	garr_betriebsmeldungen[st_config.i16_meld_startindex + 0] := fb_ton_abfrage_wt_auf_beladepos.Q;
	garr_betriebsmeldungen[st_config.i16_meld_startindex + 1] := fb_ton_warte_auf_wt_an_stopper.Q;
	garr_betriebsmeldungen[st_config.i16_meld_startindex + 2] := FALSE;
	garr_betriebsmeldungen[st_config.i16_meld_startindex + 3] := FALSE;
	garr_betriebsmeldungen[st_config.i16_meld_startindex + 4] := FALSE;
	garr_betriebsmeldungen[st_config.i16_meld_startindex + 5] := FALSE;
	garr_betriebsmeldungen[st_config.i16_meld_startindex + 6] := FALSE;
	garr_betriebsmeldungen[st_config.i16_meld_startindex + 7] := FALSE;
	garr_betriebsmeldungen[st_config.i16_meld_startindex + 8] := FALSE;
	garr_betriebsmeldungen[st_config.i16_meld_startindex + 9] := FALSE;
	garr_betriebsmeldungen[st_config.i16_meld_startindex + 10] := FALSE;
	garr_betriebsmeldungen[st_config.i16_meld_startindex + 11] := FALSE;
	garr_betriebsmeldungen[st_config.i16_meld_startindex + 12] := FALSE;
	garr_betriebsmeldungen[st_config.i16_meld_startindex + 13] := FALSE;
	garr_betriebsmeldungen[st_config.i16_meld_startindex + 14] := FALSE;
	garr_betriebsmeldungen[st_config.i16_meld_startindex + 15] := FALSE;
	garr_betriebsmeldungen[st_config.i16_meld_startindex + 16] := FALSE;
	garr_betriebsmeldungen[st_config.i16_meld_startindex + 17] := FALSE;
	garr_betriebsmeldungen[st_config.i16_meld_startindex + 18] := FALSE;
	garr_betriebsmeldungen[st_config.i16_meld_startindex + 19] := FALSE;
END_IF
END_PROGRAM

(* POU Gemeinsamkeiten17xx/WT Transport/ST_Hublift_links, ST *)
PROGRAM ST_Hublift_links
VAR_INPUT
	st_config							: struct_config;
	st_ctrl_in							: struct_ctrl_in;
	e_station_nachher_in_erlaubnis		: BOOL := FALSE;
	e_station_nachher_in_angekommen	: BOOL := FALSE;
END_VAR
VAR_IN_OUT
	st_visu							: struct_visu;
END_VAR
VAR_OUTPUT
	st_ctrl_out						: struct_ctrl_out;
	a_station_nachher_out_anforderung	: BOOL := FALSE;
	a_station_nachher_out_abgegeben	: BOOL := FALSE;
END_VAR
VAR
	fb_ton_wz						: TON;
	fb_ton_uez						: TON;
	tb_ton_wt_anwesend				: TON;
	fb_ton_quitt						: TON;
	fb_r_trig_start						: R_TRIG;
	fb_state_entry						: ST_StateEntry;
	sm_kein_wt_anwesend				: BOOL := FALSE;
	sm_keine_busverbindung			: BOOL := FALSE;
	sm_schiebetuere_nicht_geschlossen	: BOOL := FALSE;

	e_sensor_wt_anwesend			AT %I* : BOOL;
	e_sensor_wt_von_fb_eingezogen	AT %I* : BOOL;
	e_wc_state						AT%I*: BOOL;	(* 0=Data valid, 1=Data invalid *)

	e_schiebetuere_geschlossen			AT %I* : BOOL;
	a_lampe_erlaubnis_schiebetuere_oeffnen		AT %Q* : BOOL;	(* Wenn Lampe TRUE dann darf der Bediener die Schiebetüre öffnen *)
END_VAR
(* Zeiten *)
fb_ton_wz(IN:= , PT:= , Q=>  , ET=> );
fb_ton_uez(IN:= , PT:= , Q=>  , ET=> );
tb_ton_wt_anwesend(IN:=e_sensor_wt_anwesend , PT:= t#500ms, Q=>  , ET=> );
fb_ton_quitt(IN:= , PT:= t#100ms, Q=> , ET=> );

(* Flanken *)
fb_r_trig_start(CLK:=ST_Euchner_Handbedienpult.b_Taste_Power , Q=>);

(* Toplevel *)
IF fb_state_entry.i16_next_step > INIT AND fb_state_entry.i16_next_step < FEHLER THEN
	IF fb_state_entry.i16_next_step < STOP THEN
		IF st_ctrl_in.b_stop THEN
			fb_state_entry.i16_next_step := STOP;
		END_IF
	END_IF

	(* Allgemeine Fehler *)
	IF 	st_config.b_station_aktiv AND NOT st_config.b_station_in_simulation AND
		(zyl_hublift_links_lift.st_ctrl.out.b_fehler OR
		zyl_hublift_links_wt_einzug.st_ctrl.out.b_fehler OR
		zyl_hublift_links_wt_klinke.st_ctrl.out.b_fehler OR
		zyl_hublift_links_stopper.st_ctrl.out.b_fehler OR
		zyl_hublift_links_eingriffschutz.st_ctrl.out.b_fehler) THEN
			fb_state_entry.i16_next_step := FEHLER;

	(* Zylinder im Handbetrieb *)
	ELSIF gi16_betriebsart = HAND AND st_config.b_station_aktiv AND NOT st_config.b_station_in_simulation AND
		((st_visu.st_zyl.i16_nr_zyl_im_handbetrieb = zyl_hublift_links_lift.fb.st_config.i16_identnummer) OR
		(st_visu.st_zyl.i16_nr_zyl_im_handbetrieb = zyl_hublift_links_wt_einzug.fb.st_config.i16_identnummer) OR
		(st_visu.st_zyl.i16_nr_zyl_im_handbetrieb = zyl_hublift_links_wt_klinke.fb.st_config.i16_identnummer) OR
		(st_visu.st_zyl.i16_nr_zyl_im_handbetrieb = zyl_hublift_links_stopper.fb.st_config.i16_identnummer)  OR
		(st_visu.st_zyl.i16_nr_zyl_im_handbetrieb = zyl_hublift_links_eingriffschutz.fb.st_config.i16_identnummer) ) THEN
			fb_state_entry.i16_next_step := FEHLER;
	END_IF
END_IF

(* ==================================Schrittkette================================ *)
fb_state_entry(
	i16_next_step:= ,
	i16_pos:= 1,
	s_debugtext:= ,
	E=> ,
	X=> ,
	i16_step=> ,
	i16_last_step=> );

CASE fb_state_entry.i16_step OF
(*=======================================================*)
	INIT_OBJ:
		IF st_config.b_config_fertig THEN
			fb_state_entry.i16_next_step := INIT;
		END_IF

(*=======================================================*)
	INIT:
		IF fb_state_entry.E THEN
			fb_ton_wz.IN := FALSE;
			fb_ton_uez.IN	:= FALSE;
			fb_ton_quitt.IN := FALSE;
			sm_kein_wt_anwesend	:= FALSE;
			sm_keine_busverbindung := FALSE;
			sm_schiebetuere_nicht_geschlossen := FALSE;
			a_station_nachher_out_anforderung := FALSE;
			a_station_nachher_out_abgegeben := FALSE;
			a_lampe_erlaubnis_schiebetuere_oeffnen := FALSE;
			st_ctrl_out.b_fehler := FALSE;
			st_ctrl_out.b_bereit := FALSE;
			st_ctrl_out.b_fertig := FALSE;
			st_ctrl_out.b_kontroller_start := FALSE;
			zyl_hublift_links_lift.st_ctrl.in.b_einfahren := FALSE;
			zyl_hublift_links_lift.st_ctrl.in.b_ausfahren := FALSE;
			zyl_hublift_links_wt_einzug.st_ctrl.in.b_einfahren := FALSE;
			zyl_hublift_links_wt_einzug.st_ctrl.in.b_ausfahren := FALSE;
			zyl_hublift_links_wt_klinke.st_ctrl.in.b_einfahren := FALSE;
			zyl_hublift_links_wt_klinke.st_ctrl.in.b_ausfahren := FALSE;
			zyl_hublift_links_stopper.st_ctrl.in.b_einfahren := FALSE;
			zyl_hublift_links_stopper.st_ctrl.in.b_ausfahren := FALSE;
			zyl_hublift_links_eingriffschutz.st_ctrl.in.b_einfahren := FALSE;
			zyl_hublift_links_eingriffschutz.st_ctrl.in.b_ausfahren := FALSE;
		END_IF

		(*-----------------------Weiterschaltbedingungen----------------------------*)
		IF st_ctrl_in.b_init THEN
			zyl_hublift_links_lift.st_ctrl.in.b_quittieren := FALSE;
			zyl_hublift_links_wt_einzug.st_ctrl.in.b_quittieren := FALSE;
			zyl_hublift_links_wt_klinke.st_ctrl.in.b_quittieren := FALSE;
			zyl_hublift_links_stopper.st_ctrl.in.b_quittieren := FALSE;
			zyl_hublift_links_eingriffschutz.st_ctrl.in.b_quittieren := FALSE;

			IF st_config.b_station_aktiv AND NOT st_config.b_station_in_simulation AND gst_datensatz.st_md.b_wt_transport_aktiv THEN
				fb_state_entry.i16_next_step := 15;
			ELSE
				fb_state_entry.i16_next_step := BEREIT;
			END_IF
		END_IF

(*=======================================================*)
	15: (* Prüfe, ob Busverbindung vorhanden ist *)

		(*-----------------------Weiterschaltbedingungen----------------------------*)
		IF e_wc_state THEN
			sm_keine_busverbindung := TRUE;
			fb_state_entry.i16_next_step := FEHLER;
		ELSE
			fb_state_entry.i16_next_step := 18;
		END_IF

(*=======================================================*)
	18: (* Prüfe, ob Eingriffschutz geschlossen ist *)

		(*-----------------------Weiterschaltbedingungen----------------------------*)
		IF NOT e_schiebetuere_geschlossen THEN
			sm_schiebetuere_nicht_geschlossen := TRUE;
			fb_state_entry.i16_next_step := FEHLER;
		ELSE
			fb_state_entry.i16_next_step := 20;
		END_IF

(*=======================================================*)
	20: (* Initialisierung: Stopper ausfahren *)
		IF fb_state_entry.E THEN
			zyl_hublift_links_stopper.st_ctrl.in.b_ausfahren := TRUE;
		END_IF

		(*-----------------------Weiterschaltbedingungen----------------------------*)
		IF zyl_hublift_links_stopper.st_ctrl.out.b_ausgefahren THEN
			zyl_hublift_links_stopper.st_ctrl.in.b_ausfahren := FALSE;
			fb_state_entry.i16_next_step := 30;
		END_IF

(*=======================================================*)
	30: (* Initialisierung: Abfrage auf WT *)
		IF tb_ton_wt_anwesend.Q THEN
		(* WT anwesend *)
			IF zyl_hublift_links_lift.fb.e_sensor1_eingefahren THEN
			(* Hublift unten *)
				fb_state_entry.i16_next_step := 120;
			ELSE
			(* Hublift oben *)
				fb_state_entry.i16_next_step := 155;
			END_IF
		ELSE
		(* Kein WT vorhanden oder vielleicht steht einer am Stopper *)
			fb_state_entry.i16_next_step := 40;
		END_IF

(*=======================================================*)
	40: (* Initialisierung: Klinke einfahren *)
		IF fb_state_entry.E THEN
			zyl_hublift_links_wt_klinke.st_ctrl.in.b_einfahren := TRUE;
		END_IF

		(*-----------------------Weiterschaltbedingungen----------------------------*)
		IF zyl_hublift_links_wt_klinke.st_ctrl.out.b_eingefahren THEN
			zyl_hublift_links_wt_klinke.st_ctrl.in.b_einfahren := FALSE;
			IF zyl_hublift_links_lift.fb.e_sensor1_eingefahren THEN
			(* Hublift unten *)
				fb_state_entry.i16_next_step := 70;
			ELSE
			(* Hublift oben *)
				fb_state_entry.i16_next_step := 50;
			END_IF
		END_IF

(*=======================================================*)
	50: (* Initialisierung: WT-Einzug einfahren *)
		IF fb_state_entry.E THEN
			zyl_hublift_links_wt_einzug.st_ctrl.in.b_einfahren := TRUE;
		END_IF

		(*-----------------------Weiterschaltbedingungen----------------------------*)
		IF zyl_hublift_links_wt_einzug.st_ctrl.out.b_eingefahren THEN
			zyl_hublift_links_wt_einzug.st_ctrl.in.b_einfahren := FALSE;
			fb_state_entry.i16_next_step := 60;
		END_IF

(*=======================================================*)
	60: (* Initialisierung: Lift einfahren *)
		IF fb_state_entry.E THEN
			zyl_hublift_links_lift.st_ctrl.in.b_einfahren := TRUE;
		END_IF

		(*-----------------------Weiterschaltbedingungen----------------------------*)
		IF zyl_hublift_links_lift.st_ctrl.out.b_eingefahren THEN
			zyl_hublift_links_lift.st_ctrl.in.b_einfahren := FALSE;
			fb_state_entry.i16_next_step := 70;
		END_IF

(*=======================================================*)
	70: (* WT-Einzug ausfahren *)
		IF fb_state_entry.E THEN
			zyl_hublift_links_wt_einzug.st_ctrl.in.b_ausfahren := TRUE;
		END_IF

		(*-----------------------Weiterschaltbedingungen----------------------------*)
		IF zyl_hublift_links_wt_einzug.st_ctrl.out.b_ausgefahren THEN
			zyl_hublift_links_wt_einzug.st_ctrl.in.b_ausfahren := FALSE;
			fb_state_entry.i16_next_step := 80;
		END_IF

(*=======================================================*)
	80: (* Initialisierung: Stopper einfahren *)
		IF fb_state_entry.E THEN
			zyl_hublift_links_stopper.st_ctrl.in.b_einfahren := TRUE;
		END_IF

		(*-----------------------Weiterschaltbedingungen----------------------------*)
		IF zyl_hublift_links_stopper.st_ctrl.out.b_eingefahren THEN
			zyl_hublift_links_stopper.st_ctrl.in.b_einfahren := FALSE;
			fb_state_entry.i16_next_step := 90;
		END_IF

(*=======================================================*)
	90: (* Eingriffschutz ausfahren*)
		IF fb_state_entry.E THEN
			zyl_hublift_links_eingriffschutz.st_ctrl.in.b_ausfahren := TRUE;
		END_IF

		(*-----------------------Weiterschaltbedingungen----------------------------*)
		IF zyl_hublift_links_eingriffschutz.st_ctrl.out.b_ausgefahren THEN
			zyl_hublift_links_eingriffschutz.st_ctrl.in.b_ausfahren := FALSE;
			fb_state_entry.i16_next_step := BEREIT;
		END_IF

(*=======================================================*)
	BEREIT:
		IF fb_state_entry.E THEN
			st_ctrl_out.b_bereit := TRUE;
		END_IF

		(*-----------------------Weiterschaltbedingungen----------------------------*)
		IF st_config.b_station_aktiv AND NOT st_config.b_station_in_simulation AND gst_datensatz.st_md.b_wt_transport_aktiv THEN
			(* Hublift und WT Transport aktiv *)
			fb_state_entry.i16_next_step := 110;
		ELSIF NOT st_config.b_station_aktiv AND st_config.b_station_in_simulation AND gst_datensatz.st_md.b_wt_transport_aktiv THEN
			(* Simulation des Hubliftes *)
			fb_state_entry.i16_next_step := 160;
		ELSE
			;(* Hublift und WT Transport NICHT aktiv *)
		END_IF

(*=======================================================*)
	110:	(* Warte bis der WT angekommen ist *)

		(*-----------------------Weiterschaltbedingungen----------------------------*)
		IF tb_ton_wt_anwesend.Q THEN
			fb_state_entry.i16_next_step := 120;
		END_IF

(*=======================================================*)
	120: (* Klinke ausfahren -> WT einhaken*)
		IF fb_state_entry.E THEN
			zyl_hublift_links_wt_klinke.st_ctrl.in.b_ausfahren := TRUE;
		END_IF

		(*-----------------------Weiterschaltbedingungen----------------------------*)
		IF zyl_hublift_links_wt_klinke.st_ctrl.out.b_ausgefahren AND
			e_sensor_wt_anwesend THEN
			zyl_hublift_links_wt_klinke.st_ctrl.in.b_ausfahren := FALSE;
			fb_state_entry.i16_next_step := 130;
		END_IF

(*=======================================================*)
	130: (* WT-Einzug einfahren und Stopper bei Signal ausfahren *)
		IF fb_state_entry.E THEN
			zyl_hublift_links_wt_einzug.st_ctrl.in.b_einfahren := TRUE;
		END_IF

		(*-----------------------Weiterschaltbedingungen----------------------------*)
		IF 	e_sensor_wt_von_fb_eingezogen OR
			zyl_hublift_links_wt_einzug.st_ctrl.out.b_eingefahren THEN
				zyl_hublift_links_stopper.st_ctrl.in.b_ausfahren := TRUE;
				fb_state_entry.i16_next_step := 140;
		END_IF

(*=======================================================*)
	140: (* WT-Einzug ist eingefahren und Stopper ist ausgefahren *)

		(*-----------------------Weiterschaltbedingungen----------------------------*)
		IF 	zyl_hublift_links_stopper.st_ctrl.out.b_ausgefahren AND
			zyl_hublift_links_wt_einzug.st_ctrl.out.b_eingefahren AND
			e_sensor_wt_anwesend THEN
				zyl_hublift_links_stopper.st_ctrl.in.b_ausfahren := FALSE;
				zyl_hublift_links_wt_einzug.st_ctrl.in.b_einfahren := FALSE;
				fb_state_entry.i16_next_step := 150;
		END_IF

(*=======================================================*)
	150: (* WT mit Lift anheben *)
		IF fb_state_entry.E THEN
			zyl_hublift_links_lift.st_ctrl.in.b_ausfahren := TRUE;
		END_IF

		(*-----------------------Weiterschaltbedingungen----------------------------*)
		IF zyl_hublift_links_lift.st_ctrl.out.b_ausgefahren THEN
			zyl_hublift_links_lift.st_ctrl.in.b_ausfahren := FALSE;
			fb_state_entry.i16_next_step := 155;
		END_IF

(*=======================================================*)
	155: (* Warte auf Simulation oder Taste_Power *)
		IF fb_state_entry.E THEN
			a_lampe_erlaubnis_schiebetuere_oeffnen := TRUE;
		END_IF

		(*-----------------------Weiterschaltbedingungen----------------------------*)
		IF st_config.b_station_in_simulation OR
			(fb_r_trig_start.Q AND e_schiebetuere_geschlossen) THEN
			fb_state_entry.i16_next_step := 160;
		END_IF

		IF fb_state_entry.X THEN
			a_lampe_erlaubnis_schiebetuere_oeffnen := FALSE;
		END_IF

(*=======================================================*)
	160: (* Warte auf Folgestation *)
		IF fb_state_entry.E THEN
			st_ctrl_out.b_bereit := TRUE;
			a_station_nachher_out_anforderung := TRUE;
		END_IF

		(*-----------------------Weiterschaltbedingungen----------------------------*)
		IF  e_station_nachher_in_erlaubnis AND NOT fb_state_entry.E THEN
			a_station_nachher_out_anforderung := FALSE;
			IF st_config.b_station_in_simulation THEN
				fb_state_entry.i16_next_step := 180;
			ELSE
				IF e_sensor_wt_anwesend THEN
					fb_state_entry.i16_next_step := 165;
				ELSE
					fb_state_entry.i16_next_step := 190;
				END_IF
			END_IF
		END_IF

(*=======================================================*)
	165: (* Eingriffschutz einfahren*)
		IF fb_state_entry.E THEN
			zyl_hublift_links_eingriffschutz.st_ctrl.in.b_einfahren := TRUE;
		END_IF

		(*-----------------------Weiterschaltbedingungen----------------------------*)
		IF zyl_hublift_links_eingriffschutz.st_ctrl.out.b_eingefahren THEN
			zyl_hublift_links_eingriffschutz.st_ctrl.in.b_einfahren := FALSE;
			fb_state_entry.i16_next_step := 170;
		END_IF

(*=======================================================*)
	170: (* WT-Einzug ausfahren und Klinke einfahren und WT aushaken *)
		IF fb_state_entry.E THEN
			zyl_hublift_links_wt_einzug.st_ctrl.in.b_ausfahren := TRUE;
			zyl_hublift_links_wt_klinke.st_ctrl.in.b_einfahren := TRUE;
			st_ctrl_out.b_kontroller_start := TRUE;
		END_IF

		(*-----------------------Weiterschaltbedingungen----------------------------*)
		IF 	zyl_hublift_links_wt_einzug.st_ctrl.out.b_ausgefahren AND
			zyl_hublift_links_wt_klinke.st_ctrl.out.b_eingefahren
			THEN
				st_ctrl_out.b_kontroller_start := FALSE;
				zyl_hublift_links_wt_einzug.st_ctrl.in.b_ausfahren := FALSE;
				zyl_hublift_links_wt_klinke.st_ctrl.in.b_einfahren := FALSE;
				fb_state_entry.i16_next_step := 180;
		END_IF

(*=======================================================*)
	180:	(* Warte bis WT angekommen ist *)
		IF fb_state_entry.E THEN
			a_station_nachher_out_abgegeben := TRUE;
		END_IF

		(*-----------------------Weiterschaltbedingungen----------------------------*)
		IF e_station_nachher_in_angekommen THEN
			a_station_nachher_out_abgegeben := FALSE;
			IF st_config.b_station_in_simulation THEN
				fb_state_entry.i16_next_step := BEREIT;
			ELSE
				fb_state_entry.i16_next_step := 185;
			END_IF
		END_IF

(*=======================================================*)
	185: (* Eingriffschutz ausfahren*)
		IF fb_state_entry.E THEN
			zyl_hublift_links_eingriffschutz.st_ctrl.in.b_ausfahren := TRUE;
		END_IF

		(*-----------------------Weiterschaltbedingungen----------------------------*)
		IF zyl_hublift_links_eingriffschutz.st_ctrl.out.b_ausgefahren THEN
			zyl_hublift_links_eingriffschutz.st_ctrl.in.b_ausfahren := FALSE;
			fb_state_entry.i16_next_step := 190;
		END_IF

(*=======================================================*)
	190: (* Klinke einfahren*)
		IF fb_state_entry.E THEN
			zyl_hublift_links_wt_klinke.st_ctrl.in.b_einfahren := TRUE;
		END_IF

		(*-----------------------Weiterschaltbedingungen----------------------------*)
		IF zyl_hublift_links_wt_klinke.st_ctrl.out.b_eingefahren THEN
			zyl_hublift_links_wt_klinke.st_ctrl.in.b_einfahren := FALSE;
			fb_state_entry.i16_next_step := 200;
		END_IF

(*=======================================================*)
	200: (* WT-Einzug einfahren  *)
		IF fb_state_entry.E THEN
			zyl_hublift_links_wt_einzug.st_ctrl.in.b_einfahren := TRUE;
		END_IF

		(*-----------------------Weiterschaltbedingungen----------------------------*)
		IF zyl_hublift_links_wt_einzug.st_ctrl.out.b_eingefahren THEN
			zyl_hublift_links_wt_einzug.st_ctrl.in.b_einfahren := FALSE;
			fb_state_entry.i16_next_step := 210;
		END_IF

(*=======================================================*)
	210: (*  Lift einfahren *)
		IF fb_state_entry.E THEN
			zyl_hublift_links_lift.st_ctrl.in.b_einfahren := TRUE;
		END_IF

		(*-----------------------Weiterschaltbedingungen----------------------------*)
		IF zyl_hublift_links_lift.st_ctrl.out.b_eingefahren THEN
			zyl_hublift_links_lift.st_ctrl.in.b_einfahren := FALSE;
			fb_state_entry.i16_next_step := 220;
		END_IF

(*=======================================================*)
	220: (* WT-Einzug ausfahren  *)
		IF fb_state_entry.E THEN
			zyl_hublift_links_wt_einzug.st_ctrl.in.b_ausfahren := TRUE;
		END_IF

		(*-----------------------Weiterschaltbedingungen----------------------------*)
		IF zyl_hublift_links_wt_einzug.st_ctrl.out.b_ausgefahren THEN
			zyl_hublift_links_wt_einzug.st_ctrl.in.b_ausfahren := FALSE;
			fb_state_entry.i16_next_step := 230;
		END_IF

(*=======================================================*)
	230: (* Stopper einfahren *)
		IF fb_state_entry.E THEN
			zyl_hublift_links_stopper.st_ctrl.in.b_einfahren := TRUE;
		END_IF

		(*-----------------------Weiterschaltbedingungen----------------------------*)
		IF zyl_hublift_links_stopper.st_ctrl.out.b_eingefahren THEN
			zyl_hublift_links_stopper.st_ctrl.in.b_einfahren := FALSE;
			fb_state_entry.i16_next_step := BEREIT;
		END_IF

(*=======================================================*)
	FEHLER:
		IF fb_state_entry.E THEN
			st_ctrl_out.b_fehler := TRUE;
			fb_ton_quitt.IN := FALSE;
			a_station_nachher_out_anforderung := FALSE;
			a_station_nachher_out_abgegeben := FALSE;
			zyl_hublift_links_lift.st_ctrl.in.b_quittieren := FALSE;
			zyl_hublift_links_wt_einzug.st_ctrl.in.b_quittieren := FALSE;
			zyl_hublift_links_wt_klinke.st_ctrl.in.b_quittieren := FALSE;
			zyl_hublift_links_stopper.st_ctrl.in.b_quittieren := FALSE;
			zyl_hublift_links_eingriffschutz.st_ctrl.in.b_quittieren := FALSE;
		END_IF

		(*-----------------------Weiterschaltbedingungen----------------------------*)
		IF st_ctrl_in.b_quitt AND NOT fb_state_entry.E THEN
			st_ctrl_out.b_fehler := FALSE;
			zyl_hublift_links_lift.st_ctrl.in.b_quittieren := TRUE;
			zyl_hublift_links_wt_einzug.st_ctrl.in.b_quittieren := TRUE;
			zyl_hublift_links_wt_klinke.st_ctrl.in.b_quittieren := TRUE;
			zyl_hublift_links_stopper.st_ctrl.in.b_quittieren := TRUE;
			zyl_hublift_links_eingriffschutz.st_ctrl.in.b_quittieren := TRUE;
			fb_ton_quitt.IN := TRUE;
		END_IF

		IF fb_ton_quitt.Q THEN
			fb_ton_quitt.IN := FALSE;
			fb_state_entry.i16_next_step := INIT;
		END_IF

(*=======================================================*)
	STOP:
		IF fb_state_entry.E THEN
			fb_ton_quitt.IN := FALSE;
			zyl_hublift_links_lift.st_ctrl.in.b_quittieren := FALSE;
			zyl_hublift_links_wt_einzug.st_ctrl.in.b_quittieren := FALSE;
			zyl_hublift_links_wt_klinke.st_ctrl.in.b_quittieren := FALSE;
			zyl_hublift_links_stopper.st_ctrl.in.b_quittieren := FALSE;
			zyl_hublift_links_eingriffschutz.st_ctrl.in.b_quittieren := FALSE;
		END_IF

		(*-----------------------Weiterschaltbedingungen----------------------------*)
		IF st_ctrl_in.b_quitt AND NOT fb_state_entry.E THEN
			fb_ton_quitt.IN := TRUE;
			zyl_hublift_links_lift.st_ctrl.in.b_quittieren := TRUE;
			zyl_hublift_links_wt_einzug.st_ctrl.in.b_quittieren := TRUE;
			zyl_hublift_links_wt_klinke.st_ctrl.in.b_quittieren := TRUE;
			zyl_hublift_links_stopper.st_ctrl.in.b_quittieren := TRUE;
			zyl_hublift_links_eingriffschutz.st_ctrl.in.b_quittieren := TRUE;
		END_IF

		IF fb_ton_quitt.Q THEN
			fb_ton_quitt.IN := FALSE;
			fb_state_entry.i16_next_step := INIT;
		END_IF
END_CASE

fb_state_entry(
	i16_next_step:= ,
	i16_pos:= 2,
	s_debugtext:= ,
	E=> ,
	X=> , 
	i16_step=> ,
	i16_last_step=> );

IF st_config.b_config_fertig THEN
	(* Fehlermeldungen und Betriebsmeldungen ab dem Startindex in die globalen Meldungsarrays schreiben *)
	garr_stoermeldungen[st_config.i16_meld_startindex + 0] := sm_kein_wt_anwesend;
	garr_stoermeldungen[st_config.i16_meld_startindex + 1] := sm_keine_busverbindung;
	garr_stoermeldungen[st_config.i16_meld_startindex + 2] := sm_schiebetuere_nicht_geschlossen;
	garr_stoermeldungen[st_config.i16_meld_startindex + 3] := FALSE;
	garr_stoermeldungen[st_config.i16_meld_startindex + 4] := FALSE;
	garr_stoermeldungen[st_config.i16_meld_startindex + 5] := FALSE;
	garr_stoermeldungen[st_config.i16_meld_startindex + 6] := FALSE;
	garr_stoermeldungen[st_config.i16_meld_startindex + 7] := FALSE;
	garr_stoermeldungen[st_config.i16_meld_startindex + 8] := FALSE;
	garr_stoermeldungen[st_config.i16_meld_startindex + 9] := FALSE;
	garr_stoermeldungen[st_config.i16_meld_startindex + 10] := FALSE;
	garr_stoermeldungen[st_config.i16_meld_startindex + 11] := FALSE;
	garr_stoermeldungen[st_config.i16_meld_startindex + 12] := FALSE;
	garr_stoermeldungen[st_config.i16_meld_startindex + 13] := FALSE;
	garr_stoermeldungen[st_config.i16_meld_startindex + 14] := FALSE;
	garr_stoermeldungen[st_config.i16_meld_startindex + 15] := FALSE;
	garr_stoermeldungen[st_config.i16_meld_startindex + 16] := FALSE;
	garr_stoermeldungen[st_config.i16_meld_startindex + 17] := FALSE;
	garr_stoermeldungen[st_config.i16_meld_startindex + 18] := FALSE;
	garr_stoermeldungen[st_config.i16_meld_startindex + 19] := FALSE;
	
	garr_betriebsmeldungen[st_config.i16_meld_startindex + 0] := FALSE;
	garr_betriebsmeldungen[st_config.i16_meld_startindex + 1] := FALSE;
	garr_betriebsmeldungen[st_config.i16_meld_startindex + 2] := FALSE;
	garr_betriebsmeldungen[st_config.i16_meld_startindex + 3] := FALSE;
	garr_betriebsmeldungen[st_config.i16_meld_startindex + 4] := FALSE;
	garr_betriebsmeldungen[st_config.i16_meld_startindex + 5] := FALSE;
	garr_betriebsmeldungen[st_config.i16_meld_startindex + 6] := FALSE;
	garr_betriebsmeldungen[st_config.i16_meld_startindex + 7] := FALSE;
	garr_betriebsmeldungen[st_config.i16_meld_startindex + 8] := FALSE;
	garr_betriebsmeldungen[st_config.i16_meld_startindex + 9] := FALSE;
	garr_betriebsmeldungen[st_config.i16_meld_startindex + 10] := FALSE;
	garr_betriebsmeldungen[st_config.i16_meld_startindex + 11] := FALSE;
	garr_betriebsmeldungen[st_config.i16_meld_startindex + 12] := FALSE;
	garr_betriebsmeldungen[st_config.i16_meld_startindex + 13] := FALSE;
	garr_betriebsmeldungen[st_config.i16_meld_startindex + 14] := FALSE;
	garr_betriebsmeldungen[st_config.i16_meld_startindex + 15] := FALSE;
	garr_betriebsmeldungen[st_config.i16_meld_startindex + 16] := FALSE;
	garr_betriebsmeldungen[st_config.i16_meld_startindex + 17] := FALSE;
	garr_betriebsmeldungen[st_config.i16_meld_startindex + 18] := FALSE;
	garr_betriebsmeldungen[st_config.i16_meld_startindex + 19] := FALSE;
END_IF
END_PROGRAM

(* POU Maschine1700/ST_Stoerungen_Quitt_1700, ST *)
PROGRAM ST_Stoerungen_Quitt_1700
VAR_INPUT
	st_config					: struct_config;
	st_ctrl_in					: struct_ctrl_in;
END_VAR
VAR_IN_OUT
	st_visu					: struct_visu;
	st_visu_hinten				: struct_visu_hinten;
END_VAR
VAR_OUTPUT
	st_ctrl_out				: struct_ctrl_out;
	b_lampe_stoerung		: BOOL;
	b_lampe_produktion		: BOOL;
END_VAR
VAR
	fb_ton_quitt				: TON;
	b_Merker_quitt			: BOOL:=FALSE;
	fb_ton_wz				: TON;
	fb_r_trig_quittieren			: R_TRIG;
	fb_state_entry				: ST_StateEntry;

	fb_blinker				: ST_Blinker;

	bm_Maschine_in_Gst		: BOOL := FALSE;
	bm_Check		: BOOL := FALSE;
	sm_disable_auto_reset	: BOOL := FALSE;
END_VAR
(* Zeiten *)
fb_ton_quitt(IN:= , PT:= t#300ms, Q=> , ET=> );
fb_ton_wz(IN:= , PT:= t#3000ms, Q=> , ET=> );

(* Flanken *)
fb_r_trig_quittieren(CLK:= (st_visu.b_quittieren OR st_visu_hinten.out.b_quittieren) AND gi16_betriebsart <> HAND, Q=> );

(* Blinker *)
fb_blinker(
	b_start:= TRUE,
	t_taktzeit_on:=t#500ms,
	t_taktzeit_off:=t#500ms,
	b_blinker_out=> );

(* Lampen *)
b_lampe_stoerung := gi16_maschinenstatusinfo = KEIN_STATUS OR gi16_maschinenstatusinfo = STATUS_FEHLER;

b_lampe_produktion := (fb_blinker.b_blinker_out AND
					(gi16_maschinenstatusinfo = STATUS_FEHLER_QUITTIERT OR
					gi16_maschinenstatusinfo = STATUS_BETRIEBSBEREIT)) OR
					gi16_maschinenstatusinfo = STATUS_MASCHINE_ARBEITET;

bm_Check:=(
	CheckBounds_ErrCnt+
	CheckByteZeroDiv_ErrCnt+
	CheckDWordZeroDiv_ErrCnt+
	CheckRealZeroDiv_ErrCnt+
	CheckWordZeroDiv_ErrCnt+
	CheckRangeSigned_ErrCnt+
	CheckRangeUnsigned_ErrCnt) > 0 ;

(* Toplevel *)
(* Hier nur Abschaltungen welche zu sofortigem Stop führen müssen *)
IF fb_state_entry.i16_step < FEHLER AND
	(axis_virt_master.st_ctrl.out.b_fehler OR
	axis_bestueckachse.st_ctrl.out.b_fehler OR
	axis_z_achse.st_ctrl.out.b_fehler OR
	axis_y_achse.st_ctrl.out.b_fehler OR
	ST_TouchProbe.st_ctrl_out.b_fehler OR
	(axis_bandeinzug_achse.st_ctrl.out.b_fehler AND gst_datensatz.st_wkz.i16_typ_bandeinzug = SERVO) OR
	bandspruehoeler.st_ctrl.out.b_fehler OR
	(bandeinzug_kontroller.st_ctrl.out.b_fehler AND gst_datensatz.st_wkz.i16_typ_bandeinzug = BANDWECHSLER_V2) OR
	bandwechsel_kontroller.st_ctrl.out.b_fehler OR
	wkz_absicherung.st_ctrl.out.b_fehler OR
	wt_transport_kontroller.st_ctrl.out.b_fehler OR
	balluff_tag_reader.st_ctrl.out.b_fehler OR
	haspel_kontroller.st_ctrl.out.b_fehler OR
	bbgen.st_ctrl.out.b_fehler OR
	wartung.st_ctrl.out.b_fehler OR
	betriebsfreigaben.st_ctrl.out.b_fehler OR
	einpresskraft_kontroller.st_ctrl.out.b_fehler OR
	safety.st_ctrl.out.b_fehler OR
	edit_mfps.st_ctrl.out.b_fehler OR
	Lesen_Schreiben_Tag.st_ctrl.out.b_fehler OR
	Service.st_ctrl.out.b_fehler OR
	axis_transport_wt_achse.st_ctrl.out.b_fehler)
	THEN
		fb_state_entry.i16_next_step := FEHLER;
END_IF

(* Prüfe ob BA = Hand -> Stoppe Abläufe *)
IF  fb_state_entry.i16_step > INIT  AND fb_state_entry.i16_step < FEHLER  AND gi16_betriebsart = HAND THEN
	fb_state_entry.i16_next_step := FEHLER;
END_IF

(* ======================================Schrittkette======================================== *)
fb_state_entry(
	i16_next_step:= ,
	i16_pos:= 1,
	s_debugtext:= ,
	E=> ,
	X=> ,
	i16_step=> ,
	i16_last_step=> );

CASE fb_state_entry.i16_step OF
(*=======================================================*)
	INIT_OBJ:
		IF st_config.b_config_fertig THEN
			fb_state_entry.i16_next_step := FEHLER;
		END_IF

(*=======================================================*)
	INIT:
		IF fb_state_entry.E THEN
			gi16_maschinenstatusinfo := STATUS_FEHLER_QUITTIERT;
			fb_ton_quitt.IN := FALSE;
			UPS.st_ctrl.in.b_quitt := FALSE;
			betriebsfreigaben.st_ctrl.in.b_quitt := FALSE;
			bandeinzug_kontroller.st_ctrl.in.b_quitt := FALSE;
			bandwechsel_kontroller.st_ctrl.in.b_quitt := FALSE;
			axis_virt_master.st_ctrl.in.b_quitt := FALSE;
			axis_bestueckachse.st_ctrl.in.b_quitt := FALSE;
			axis_y_achse.st_ctrl.in.b_quitt := FALSE;
			axis_z_achse.st_ctrl.in.b_quitt := FALSE;
			ST_TouchProbe.st_ctrl_in.b_quitt := FALSE;
			axis_bandeinzug_achse.st_ctrl.in.b_quitt := FALSE;
			bandspruehoeler.st_ctrl.in.b_quitt := FALSE;
			haspel_kontroller.st_ctrl.in.b_quitt := FALSE;
			hublift_links.st_ctrl.in.b_quitt := FALSE;
			hublift_rechts.st_ctrl.in.b_quitt := FALSE;
			wt_transport_kontroller.st_ctrl.in.b_quitt := FALSE;
			wkz_absicherung.st_ctrl.in.b_quitt := FALSE;
			stueckzahlen.st_ctrl.in.b_quitt := FALSE;
			balluff_tag_reader.st_ctrl.in.b_quitt := FALSE;
			bbgen.st_ctrl.in.b_quitt := FALSE;
			wartung.st_ctrl.in.b_quitt := FALSE;
			einpresskraft_kontroller.st_ctrl.in.b_quitt := FALSE;
			safety.st_ctrl.in.b_quitt := FALSE;
			edit_mfps.st_ctrl.in.b_quitt := FALSE;
			routing_backpanel.st_ctrl.in.b_quitt := FALSE;
			routing_nachbarpc.st_ctrl.in.b_quitt := FALSE;
			bm_Maschine_in_Gst := FALSE;
			Lesen_Schreiben_Tag.st_ctrl.in.b_quitt := FALSE;
			Service.st_ctrl.in.b_quitt := FALSE;
			ST_TippTasten.b_initialisierungsphase := TRUE;
			sm_disable_auto_reset := FALSE;
			axis_transport_wt_achse.st_ctrl.in.b_quitt := FALSE;
		END_IF

		(*-----------------------Weiterschaltbedingungen----------------------------*)
		IF safety.st_ctrl.out.b_bereit THEN
			fb_state_entry.i16_next_step := 11;
		END_IF

(*=======================================================*)
	11:
		IF fb_state_entry.E THEN
			axis_virt_master.st_ctrl.in.b_preinit := TRUE;
		END_IF

		(*-----------------------Weiterschaltbedingungen----------------------------*)
		IF axis_virt_master.st_ctrl.out.b_prebereit  THEN
			axis_virt_master.st_ctrl.in.b_preinit := FALSE;
			fb_state_entry.i16_next_step := 12;
		END_IF

(*=======================================================*)
	12:
		IF fb_state_entry.E THEN
			axis_z_achse.st_ctrl.in.b_preinit := TRUE;
		END_IF

		(*-----------------------Weiterschaltbedingungen----------------------------*)
		IF axis_z_achse.st_ctrl.out.b_prebereit  THEN
			axis_z_achse.st_ctrl.in.b_preinit := FALSE;
			fb_state_entry.i16_next_step := 13;
		END_IF

(*=======================================================*)
	13:
		IF fb_state_entry.E THEN
			axis_y_achse.st_ctrl.in.b_preinit := TRUE;
		END_IF

		(*-----------------------Weiterschaltbedingungen----------------------------*)
		IF axis_y_achse.st_ctrl.out.b_prebereit  THEN
			axis_y_achse.st_ctrl.in.b_preinit := FALSE;
			fb_state_entry.i16_next_step := 14;
		END_IF

(*=======================================================*)
	14:
		CASE gst_datensatz.st_wkz.i16_typ_bandeinzug OF
			BANDWECHSLER_V2:
				fb_state_entry.i16_next_step := 15;
			SERVO:
				IF fb_state_entry.E THEN
					axis_bandeinzug_achse.st_ctrl.in.b_preinit := TRUE;
				END_IF

				(*-----------------------Weiterschaltbedingungen----------------------------*)
				IF axis_bandeinzug_achse.st_ctrl.out.b_prebereit  THEN
					axis_bandeinzug_achse.st_ctrl.in.b_preinit := FALSE;
					fb_state_entry.i16_next_step := 15;
				END_IF
		END_CASE

(*=======================================================*)
	15:
		IF fb_state_entry.E THEN
			axis_bestueckachse.st_ctrl.in.b_preinit := TRUE;
		END_IF

		(*-----------------------Weiterschaltbedingungen----------------------------*)
		IF axis_bestueckachse.st_ctrl.out.b_prebereit  THEN
			axis_bestueckachse.st_ctrl.in.b_preinit := FALSE;
			fb_state_entry.i16_next_step := 16;
		END_IF

(*=======================================================*)
	16:
		(*Wenn die Bestückachse nicht in einem bestimmten Bereich steht, dann muss sie von Hand
		    freigefahren werden. Außer es ist die Nocke auf 0,0 gestellt*)
		IF	gst_datensatz.st_wkz.nockenschaltwerk_bestueckachse.arr_nocken[SP_DISABLE_AUTO_RESET].r_cam_begin = 0 AND
			gst_datensatz.st_wkz.nockenschaltwerk_bestueckachse.arr_nocken[SP_DISABLE_AUTO_RESET].r_cam_end = 0 THEN
				fb_state_entry.i16_next_step := 17;
		ELSE
			IF gst_datensatz.st_wkz.nockenschaltwerk_bestueckachse.arr_nocken[SP_DISABLE_AUTO_RESET].r_cam_begin > gst_datensatz.st_wkz.nockenschaltwerk_bestueckachse.arr_nocken[SP_DISABLE_AUTO_RESET].r_cam_end THEN
				IF bestueckachse.NcToPlc.ModuloActPos > gst_datensatz.st_wkz.nockenschaltwerk_bestueckachse.arr_nocken[SP_DISABLE_AUTO_RESET].r_cam_begin OR
					bestueckachse.NcToPlc.ModuloActPos < gst_datensatz.st_wkz.nockenschaltwerk_bestueckachse.arr_nocken[SP_DISABLE_AUTO_RESET].r_cam_end THEN
					sm_disable_auto_reset := TRUE;
					fb_state_entry.i16_next_step := FEHLER;
				ELSE
					fb_state_entry.i16_next_step := 17;
				END_IF
			ELSE
				IF bestueckachse.NcToPlc.ModuloActPos > gst_datensatz.st_wkz.nockenschaltwerk_bestueckachse.arr_nocken[SP_DISABLE_AUTO_RESET].r_cam_begin AND
					bestueckachse.NcToPlc.ModuloActPos < gst_datensatz.st_wkz.nockenschaltwerk_bestueckachse.arr_nocken[SP_DISABLE_AUTO_RESET].r_cam_end THEN
					sm_disable_auto_reset := TRUE;
					fb_state_entry.i16_next_step := FEHLER;
				ELSE
					fb_state_entry.i16_next_step := 17;
				END_IF
			END_IF
		END_IF
(*=======================================================*)
	17:
		(*-----------------------Weiterschaltbedingungen----------------------------*)
		IF 	gst_datensatz.st_md.b_anwahl_transport_achse  THEN
			fb_state_entry.i16_next_step := 18;
		ELSE
			fb_state_entry.i16_next_step := 20;
		END_IF

(*=======================================================*)
	18:
		IF fb_state_entry.E THEN
			axis_transport_wt_achse.st_ctrl.in.b_preinit := TRUE;
		END_IF

		(*-----------------------Weiterschaltbedingungen----------------------------*)
		IF axis_transport_wt_achse.st_ctrl.out.b_prebereit  THEN
			axis_transport_wt_achse.st_ctrl.in.b_preinit := FALSE;
			fb_state_entry.i16_next_step := 20;
		END_IF

(*=======================================================*)
	20:
		IF fb_state_entry.E THEN
			haspel_kontroller.st_ctrl.in.b_init := TRUE;
			bandspruehoeler.st_ctrl.in.b_init := TRUE;
			wkz_absicherung.st_ctrl.in.b_init := TRUE;
			stueckzahlen.st_ctrl.in.b_init := TRUE;
			(*balluff_tag_reader.st_ctrl.in.b_init := TRUE;*)
			einpresskraft_kontroller.st_ctrl.in.b_init := TRUE;
			edit_mfps.st_ctrl.in.b_init := TRUE;
		END_IF

		(*-----------------------Weiterschaltbedingungen----------------------------*)
		IF 	haspel_kontroller.st_ctrl.out.b_bereit  AND
			bandspruehoeler.st_ctrl.out.b_bereit  AND
			wkz_absicherung.st_ctrl.out.b_bereit AND
			einpresskraft_kontroller.st_ctrl.out.b_bereit AND
			balluff_tag_reader.st_ctrl.out.b_bereit AND
			edit_mfps.st_ctrl.out.b_bereit
			THEN
				haspel_kontroller.st_ctrl.in.b_init := FALSE;
				bandspruehoeler.st_ctrl.in.b_init := FALSE;
				wkz_absicherung.st_ctrl.in.b_init := FALSE;
				stueckzahlen.st_ctrl.in.b_init := FALSE;
				(*balluff_tag_reader.st_ctrl.in.b_init := FALSE;*)
				einpresskraft_kontroller.st_ctrl.in.b_init := FALSE;
				edit_mfps.st_ctrl.in.b_init := FALSE;
				fb_state_entry.i16_next_step := 30;
		END_IF

(*=======================================================*)
	30:
		CASE gst_datensatz.st_wkz.i16_typ_bandeinzug OF
			BANDWECHSLER_V2:
				IF fb_state_entry.E THEN
					bandeinzug_kontroller.st_ctrl.in.b_init := TRUE;
				END_IF
		
				(*-----------------------Weiterschaltbedingungen----------------------------*)
				IF bandeinzug_kontroller.st_ctrl.out.b_bereit THEN
					bandeinzug_kontroller.st_ctrl.in.b_init := FALSE;
					fb_state_entry.i16_next_step := 40;
				END_IF
			SERVO:
				fb_state_entry.i16_next_step := 40;
		END_CASE

(*=======================================================*)
	40:
		IF fb_state_entry.E THEN
			bandwechsel_kontroller.st_ctrl.in.b_init := TRUE;
		END_IF

		(*-----------------------Weiterschaltbedingungen----------------------------*)
		IF bandwechsel_kontroller.st_ctrl.out.b_bereit THEN
			bandwechsel_kontroller.st_ctrl.in.b_init := FALSE;
			fb_state_entry.i16_next_step := 50;
		END_IF

(*=======================================================*)
	50:
		IF fb_state_entry.E THEN
			axis_bestueckachse.st_ctrl.in.b_init := TRUE;
		END_IF

		(*-----------------------Weiterschaltbedingungen----------------------------*)
		IF axis_bestueckachse.st_ctrl.out.b_bereit  THEN
			axis_bestueckachse.st_ctrl.in.b_init := FALSE;
			fb_state_entry.i16_next_step := 60;
		END_IF

(*=======================================================*)
	60:
		CASE gst_datensatz.st_wkz.i16_typ_bandeinzug OF
			BANDWECHSLER_V2:
				IF fb_state_entry.E THEN
					axis_z_achse.st_ctrl.in.b_init := TRUE;
					axis_y_achse.st_ctrl.in.b_init := TRUE;
					axis_transport_wt_achse.st_ctrl.in.b_init := gst_datensatz.st_md.b_anwahl_transport_achse;
				END_IF
		
				(*-----------------------Weiterschaltbedingungen----------------------------*)
				IF 	axis_z_achse.st_ctrl.out.b_bereit AND
					axis_y_achse.st_ctrl.out.b_bereit AND
					(axis_transport_wt_achse.st_ctrl.out.b_bereit OR NOT gst_datensatz.st_md.b_anwahl_transport_achse)
					THEN
						axis_z_achse.st_ctrl.in.b_init := FALSE;
						axis_y_achse.st_ctrl.in.b_init := FALSE;
						axis_transport_wt_achse.st_ctrl.in.b_init := FALSE;
						fb_state_entry.i16_next_step := 70;
				END_IF
			SERVO:
				IF fb_state_entry.E THEN
					axis_z_achse.st_ctrl.in.b_init := TRUE;
					axis_y_achse.st_ctrl.in.b_init := TRUE;
					axis_bandeinzug_achse.st_ctrl.in.b_init := TRUE;
				END_IF
		
				(*-----------------------Weiterschaltbedingungen----------------------------*)
				IF 	axis_z_achse.st_ctrl.out.b_bereit AND
					axis_y_achse.st_ctrl.out.b_bereit AND
					axis_bandeinzug_achse.st_ctrl.out.b_bereit
					THEN
						axis_z_achse.st_ctrl.in.b_init := FALSE;
						axis_y_achse.st_ctrl.in.b_init := FALSE;
						fb_state_entry.i16_next_step := 70;
				END_IF
		END_CASE

(*=======================================================*)
	70:
		IF fb_state_entry.E THEN
			axis_virt_master.st_ctrl.in.b_init := TRUE;
		END_IF

		(*-----------------------Weiterschaltbedingungen----------------------------*)
		IF axis_virt_master.st_ctrl.out.b_bereit  THEN
			axis_virt_master.st_ctrl.in.b_init := FALSE;
			fb_state_entry.i16_next_step := 80;
		END_IF

(*=======================================================*)
	80:
		IF fb_state_entry.E THEN
			hublift_links.st_ctrl.in.b_init := TRUE;
			hublift_rechts.st_ctrl.in.b_init := TRUE;
			wt_transport_kontroller.st_ctrl.in.b_init := TRUE;
			ST_TouchProbe.st_ctrl_in.b_init := TRUE;
		END_IF

		(*-----------------------Weiterschaltbedingungen----------------------------*)
		IF hublift_links.st_ctrl.out.b_bereit AND hublift_rechts.st_ctrl.out.b_bereit AND wt_transport_kontroller.st_ctrl.out.b_bereit AND
			ST_TouchProbe.st_ctrl_out.b_bereit THEN
			hublift_links.st_ctrl.in.b_init := FALSE;
			hublift_rechts.st_ctrl.in.b_init := FALSE;
			wt_transport_kontroller.st_ctrl.in.b_init := FALSE;
			ST_TouchProbe.st_ctrl_in.b_init := FALSE;
			fb_state_entry.i16_next_step := BEREIT;
		END_IF

(*=======================================================*)
	BEREIT:
		IF fb_state_entry.E THEN
			ST_TippTasten.b_initialisierungsphase  := FALSE;
			(* Setze Maschinenstatus *)
			bm_Maschine_in_Gst := TRUE;
		END_IF

		(*Beim Einfädeln muss der Status geändert werden, damit nicht
		ständig neue Maschinendaten erzeugt werden*)
		IF ST_TippTasten.b_einfaedeln_aktiv THEN
			gi16_maschinenstatusinfo := STATUS_MASCHINE_ARBEITET;
		ELSE
			gi16_maschinenstatusinfo := STATUS_BETRIEBSBEREIT;
		END_IF

		(*-----------------------Weiterschaltbedingungen----------------------------*)
		IF NOT wt_transport_kontroller.st_ctrl.out.b_fertig THEN
			bm_Maschine_in_Gst := FALSE;
			fb_state_entry.i16_next_step := 110;
		END_IF

(*=======================================================*)
	110: (* Produktion *)
		IF fb_state_entry.E THEN
			gi16_maschinenstatusinfo := STATUS_MASCHINE_ARBEITET;
		END_IF

		(*-----------------------Weiterschaltbedingungen----------------------------*)
		IF wt_transport_kontroller.st_ctrl.out.b_fertig THEN
			fb_state_entry.i16_next_step := BEREIT;
		END_IF

(*=======================================================*)
	FEHLER:
		IF fb_state_entry.E THEN
			gi16_maschinenstatusinfo := STATUS_FEHLER;
			bm_Maschine_in_Gst := FALSE;
			ST_TippTasten.b_initialisierungsphase  := FALSE;
			fb_ton_quitt.IN := FALSE;
			fb_ton_wz.IN:=FALSE;
			s_alte_artikelnummer := '';

			(* Schlecht Stueckzahl erhöhen *)
			IF fb_state_entry.i16_last_step = 110 THEN
				stueckzahlen.st_ctrl.in.b_schlechtteil_produziert := TRUE;
			END_IF

			UPS.st_ctrl.in.b_quitt := FALSE;
			betriebsfreigaben.st_ctrl.in.b_quitt := FALSE;
			bandeinzug_kontroller.st_ctrl.in.b_quitt := FALSE;
			bandwechsel_kontroller.st_ctrl.in.b_quitt := FALSE;
			axis_virt_master.st_ctrl.in.b_quitt := FALSE;
			axis_bestueckachse.st_ctrl.in.b_quitt := FALSE;
			axis_y_achse.st_ctrl.in.b_quitt := FALSE;
			axis_z_achse.st_ctrl.in.b_quitt := FALSE;
			ST_TouchProbe.st_ctrl_in.b_quitt := FALSE;
			axis_bandeinzug_achse.st_ctrl.in.b_quitt := FALSE;
			bandspruehoeler.st_ctrl.in.b_quitt := FALSE;
			haspel_kontroller.st_ctrl.in.b_quitt := FALSE;
			hublift_links.st_ctrl.in.b_quitt := FALSE;
			hublift_rechts.st_ctrl.in.b_quitt := FALSE;
			wt_transport_kontroller.st_ctrl.in.b_quitt := FALSE;
			wkz_absicherung.st_ctrl.in.b_quitt := FALSE;
			stueckzahlen.st_ctrl.in.b_quitt := FALSE;
			balluff_tag_reader.st_ctrl.in.b_quitt := FALSE;
			bbgen.st_ctrl.in.b_quitt := FALSE;
			wartung.st_ctrl.in.b_quitt := FALSE;
			einpresskraft_kontroller.st_ctrl.in.b_quitt := FALSE;
			safety.st_ctrl.in.b_quitt := FALSE;
			edit_mfps.st_ctrl.in.b_quitt := FALSE;
			routing_backpanel.st_ctrl.in.b_quitt := FALSE;
			routing_nachbarpc.st_ctrl.in.b_quitt := FALSE;
			Lesen_Schreiben_Tag.st_ctrl.in.b_quitt := FALSE;
			Service.st_ctrl.in.b_quitt := FALSE;
			axis_transport_wt_achse.st_ctrl.in.b_quitt := FALSE;

			axis_virt_master.st_ctrl.in.b_preinit := FALSE;
			axis_bestueckachse.st_ctrl.in.b_preinit := FALSE;
			axis_y_achse.st_ctrl.in.b_preinit := FALSE;
			axis_z_achse.st_ctrl.in.b_preinit := FALSE;
			axis_bandeinzug_achse.st_ctrl.in.b_preinit := FALSE;
			axis_transport_wt_achse.st_ctrl.in.b_preinit := FALSE;

			bandeinzug_kontroller.st_ctrl.in.b_init := FALSE;
			bandwechsel_kontroller.st_ctrl.in.b_init := FALSE;
			axis_virt_master.st_ctrl.in.b_init := FALSE;
			axis_bestueckachse.st_ctrl.in.b_init := FALSE;
			axis_y_achse.st_ctrl.in.b_init := FALSE;
			axis_z_achse.st_ctrl.in.b_init := FALSE;
			ST_TouchProbe.st_ctrl_in.b_init := FALSE;
			axis_bandeinzug_achse.st_ctrl.in.b_init := FALSE;
			bandspruehoeler.st_ctrl.in.b_init := FALSE;
			haspel_kontroller.st_ctrl.in.b_init := FALSE;
			hublift_links.st_ctrl.in.b_init := FALSE;
			hublift_rechts.st_ctrl.in.b_init := FALSE;
			wt_transport_kontroller.st_ctrl.in.b_init := FALSE;
			wkz_absicherung.st_ctrl.in.b_init := FALSE;
			stueckzahlen.st_ctrl.in.b_init := FALSE;
			(*balluff_tag_reader.st_ctrl.in.b_init := FALSE;*)
			edit_mfps.st_ctrl.in.b_init := FALSE;
			axis_transport_wt_achse.st_ctrl.in.b_init := FALSE;
		END_IF

		(* Fehlerhandling: was soll bei welchem Fehler passieren? *)
		IF 	NOT fb_ton_quitt.IN THEN
			(* Stoppe/Halte Komponenten an *)
			bandeinzug_kontroller.st_ctrl.in.b_stop := TRUE;
			bandwechsel_kontroller.st_ctrl.in.b_stop := TRUE;
			bandspruehoeler.st_ctrl.in.b_stop := TRUE;
			(*haspel_kontroller.st_ctrl.in.b_stop := TRUE;*)
			hublift_links.st_ctrl.in.b_stop := TRUE;
			hublift_rechts.st_ctrl.in.b_stop := TRUE;
			wt_transport_kontroller.st_ctrl.in.b_stop := TRUE;
			stueckzahlen.st_ctrl.in.b_stop := TRUE;
			balluff_tag_reader.st_ctrl.in.b_stop := TRUE;
			edit_mfps.st_ctrl.in.b_stop := TRUE;

			(* Diese Fehler führt zum "Stop" in der Maschine *)
			IF safety.st_ctrl.out.b_fehler THEN
				axis_virt_master.st_ctrl.in.b_stop := TRUE;
				axis_bestueckachse.st_ctrl.in.b_stop := TRUE;
				axis_z_achse.st_ctrl.in.b_stop := TRUE;
				axis_y_achse.st_ctrl.in.b_stop := TRUE;
				axis_bandeinzug_achse.st_ctrl.in.b_stop := TRUE;
				axis_transport_wt_achse.st_ctrl.in.b_stop := TRUE;
				axis_virt_master.st_ctrl.in.b_halt := FALSE;
				axis_bestueckachse.st_ctrl.in.b_halt := FALSE;
				axis_z_achse.st_ctrl.in.b_halt := FALSE;
				axis_y_achse.st_ctrl.in.b_halt := FALSE;
				axis_bandeinzug_achse.st_ctrl.in.b_halt := FALSE;
				axis_transport_wt_achse.st_ctrl.in.b_halt := FALSE;
			ELSE
				axis_virt_master.st_ctrl.in.b_halt := TRUE;
				axis_bestueckachse.st_ctrl.in.b_halt := TRUE;
				axis_z_achse.st_ctrl.in.b_halt := TRUE;
				axis_y_achse.st_ctrl.in.b_halt := TRUE;
				axis_bandeinzug_achse.st_ctrl.in.b_halt := TRUE;
				axis_transport_wt_achse.st_ctrl.in.b_halt := TRUE;
				axis_virt_master.st_ctrl.in.b_stop := FALSE;
				axis_bestueckachse.st_ctrl.in.b_stop := FALSE;
				axis_z_achse.st_ctrl.in.b_stop := FALSE;
				axis_y_achse.st_ctrl.in.b_stop := FALSE;
				axis_bandeinzug_achse.st_ctrl.in.b_stop := FALSE;
				axis_transport_wt_achse.st_ctrl.in.b_stop := FALSE;
			END_IF
		END_IF

		(*-----------------------Weiterschaltbedingungen----------------------------*)
		IF 	fb_r_trig_quittieren.Q THEN
			fb_ton_wz.IN:=TRUE;
			b_Merker_quitt:=TRUE;
		END_IF
		IF 	(b_Merker_quitt AND ST_Betriebsfreigaben.e_druckwaechter) OR
			fb_ton_wz.Q THEN
			fb_ton_wz.IN:=FALSE;
			b_Merker_quitt:=FALSE;
			fb_ton_quitt.IN := TRUE;
			(* QUITT *)
			UPS.st_ctrl.in.b_quitt := TRUE;
			betriebsfreigaben.st_ctrl.in.b_quitt := TRUE;
			bandeinzug_kontroller.st_ctrl.in.b_quitt := TRUE;
			bandwechsel_kontroller.st_ctrl.in.b_quitt := TRUE;
			axis_virt_master.st_ctrl.in.b_quitt := TRUE;
			axis_bestueckachse.st_ctrl.in.b_quitt := TRUE;
			axis_y_achse.st_ctrl.in.b_quitt := TRUE;
			axis_z_achse.st_ctrl.in.b_quitt := TRUE;
			ST_TouchProbe.st_ctrl_in.b_quitt := TRUE;
			axis_bandeinzug_achse.st_ctrl.in.b_quitt := TRUE;
			bandspruehoeler.st_ctrl.in.b_quitt := TRUE;
			haspel_kontroller.st_ctrl.in.b_quitt := TRUE;
			hublift_links.st_ctrl.in.b_quitt := TRUE;
			hublift_rechts.st_ctrl.in.b_quitt := TRUE;
			wt_transport_kontroller.st_ctrl.in.b_quitt := TRUE;
			wkz_absicherung.st_ctrl.in.b_quitt := TRUE;
			stueckzahlen.st_ctrl.in.b_quitt := TRUE;
			balluff_tag_reader.st_ctrl.in.b_quitt := TRUE;
			bbgen.st_ctrl.in.b_quitt := TRUE;
			wartung.st_ctrl.in.b_quitt := TRUE;
			einpresskraft_kontroller.st_ctrl.in.b_quitt := TRUE;
			safety.st_ctrl.in.b_quitt := TRUE;
			edit_mfps.st_ctrl.in.b_quitt := TRUE;
			routing_backpanel.st_ctrl.in.b_quitt := TRUE;
			routing_nachbarpc.st_ctrl.in.b_quitt := TRUE;
			Lesen_Schreiben_Tag.st_ctrl.in.b_quitt := TRUE;
			Service.st_ctrl.in.b_quitt := TRUE;
			axis_transport_wt_achse.st_ctrl.in.b_quitt := TRUE;
			(* STOP *)
			bandeinzug_kontroller.st_ctrl.in.b_stop := FALSE;
			bandwechsel_kontroller.st_ctrl.in.b_stop := FALSE;
			axis_virt_master.st_ctrl.in.b_stop := FALSE;
			axis_bestueckachse.st_ctrl.in.b_stop := FALSE;
			axis_y_achse.st_ctrl.in.b_stop := FALSE;
			axis_z_achse.st_ctrl.in.b_stop := FALSE;
			axis_bandeinzug_achse.st_ctrl.in.b_stop := FALSE;
			bandspruehoeler.st_ctrl.in.b_stop := FALSE;
			haspel_kontroller.st_ctrl.in.b_stop := FALSE;
			hublift_links.st_ctrl.in.b_stop := FALSE;
			hublift_rechts.st_ctrl.in.b_stop := FALSE;
			wt_transport_kontroller.st_ctrl.in.b_stop := FALSE;
			wkz_absicherung.st_ctrl.in.b_stop := FALSE;
			stueckzahlen.st_ctrl.in.b_stop := FALSE;
			balluff_tag_reader.st_ctrl.in.b_stop := FALSE;
			edit_mfps.st_ctrl.in.b_stop := FALSE;
			axis_transport_wt_achse.st_ctrl.in.b_stop := FALSE;
			(* HALT - nur Achsen *)
			axis_virt_master.st_ctrl.in.b_halt := FALSE;
			axis_bestueckachse.st_ctrl.in.b_halt := FALSE;
			axis_y_achse.st_ctrl.in.b_halt := FALSE;
			axis_z_achse.st_ctrl.in.b_halt := FALSE;
			axis_bandeinzug_achse.st_ctrl.in.b_halt := FALSE;
			axis_transport_wt_achse.st_ctrl.in.b_halt := FALSE;
		END_IF

		IF fb_ton_quitt.Q THEN
			IF (gi16_betriebsart = AUTO OR gi16_betriebsart = TIPPEN) THEN
				fb_state_entry.i16_next_step := INIT;
			END_IF
		END_IF
END_CASE

fb_state_entry(
	i16_next_step:= ,
	i16_pos:= 2,
	s_debugtext:= ,
	E=> ,
	X=> , 
	i16_step=> ,
	i16_last_step=> );


(*Beim Einfädel Meldung zurücksetzen*)
IF	ST_TippTasten.b_einfaedeln_aktiv THEN
	bm_Maschine_in_Gst := FALSE;
END_IF

IF st_config.b_config_fertig THEN
	(* Fehlermeldungen und Betriebsmeldungen ab dem Startindex in die globalen Meldungsarrays schreiben *)
	garr_stoermeldungen[st_config.i16_meld_startindex + 0] := sm_disable_auto_reset;
	garr_stoermeldungen[st_config.i16_meld_startindex + 1] := FALSE;
	garr_stoermeldungen[st_config.i16_meld_startindex + 2] := FALSE;
	garr_stoermeldungen[st_config.i16_meld_startindex + 3] := FALSE;
	garr_stoermeldungen[st_config.i16_meld_startindex + 4] := FALSE;
	garr_stoermeldungen[st_config.i16_meld_startindex + 5] := FALSE;
	garr_stoermeldungen[st_config.i16_meld_startindex + 6] := FALSE;
	garr_stoermeldungen[st_config.i16_meld_startindex + 7] := FALSE;
	garr_stoermeldungen[st_config.i16_meld_startindex + 8] := FALSE;
	garr_stoermeldungen[st_config.i16_meld_startindex + 9] := FALSE;
	garr_stoermeldungen[st_config.i16_meld_startindex + 10] := FALSE;
	garr_stoermeldungen[st_config.i16_meld_startindex + 11] := FALSE;
	garr_stoermeldungen[st_config.i16_meld_startindex + 12] := FALSE;
	garr_stoermeldungen[st_config.i16_meld_startindex + 13] := FALSE;
	garr_stoermeldungen[st_config.i16_meld_startindex + 14] := FALSE;
	garr_stoermeldungen[st_config.i16_meld_startindex + 15] := FALSE;
	garr_stoermeldungen[st_config.i16_meld_startindex + 16] := FALSE;
	garr_stoermeldungen[st_config.i16_meld_startindex + 17] := FALSE;
	garr_stoermeldungen[st_config.i16_meld_startindex + 18] := FALSE;
	garr_stoermeldungen[st_config.i16_meld_startindex + 19] := FALSE;
	
	garr_betriebsmeldungen[st_config.i16_meld_startindex + 0] := bm_Maschine_in_Gst;
	garr_betriebsmeldungen[st_config.i16_meld_startindex + 1] := bm_Check;
	garr_betriebsmeldungen[st_config.i16_meld_startindex + 2] := FALSE;
	garr_betriebsmeldungen[st_config.i16_meld_startindex + 3] := FALSE;
	garr_betriebsmeldungen[st_config.i16_meld_startindex + 4] := FALSE;
	garr_betriebsmeldungen[st_config.i16_meld_startindex + 5] := FALSE;
	garr_betriebsmeldungen[st_config.i16_meld_startindex + 6] := FALSE;
	garr_betriebsmeldungen[st_config.i16_meld_startindex + 7] := FALSE;
	garr_betriebsmeldungen[st_config.i16_meld_startindex + 8] := FALSE;
	garr_betriebsmeldungen[st_config.i16_meld_startindex + 9] := FALSE;
	garr_betriebsmeldungen[st_config.i16_meld_startindex + 10] := FALSE;
	garr_betriebsmeldungen[st_config.i16_meld_startindex + 11] := FALSE;
	garr_betriebsmeldungen[st_config.i16_meld_startindex + 12] := FALSE;
	garr_betriebsmeldungen[st_config.i16_meld_startindex + 13] := FALSE;
	garr_betriebsmeldungen[st_config.i16_meld_startindex + 14] := FALSE;
	garr_betriebsmeldungen[st_config.i16_meld_startindex + 15] := FALSE;
	garr_betriebsmeldungen[st_config.i16_meld_startindex + 16] := FALSE;
	garr_betriebsmeldungen[st_config.i16_meld_startindex + 17] := FALSE;
	garr_betriebsmeldungen[st_config.i16_meld_startindex + 18] := FALSE;
	garr_betriebsmeldungen[st_config.i16_meld_startindex + 19] := FALSE;
END_IF
END_PROGRAM

(* POU Gemeinsamkeiten17xx/Haspel/Mehrfach/ST_Haspel_Kontroller_2H, ST *)
PROGRAM ST_Haspel_Kontroller_2H
VAR_INPUT
	t_abschaltzeit_motor			: TIME;
	b_drehrichtung_antrieb_links	: BOOL;
	st_config						: struct_config;
	e_druckwaechter				: BOOL;
	e_steuerung_ein				: BOOL;
	st_ctrl_in						: struct_ctrl_in;
	haspel1_ctrl_in				: struct_ctrl_out;
	haspel2_ctrl_in				: struct_ctrl_out;
END_VAR
VAR_IN_OUT
	st_visu						: struct_visu;
END_VAR
VAR_OUTPUT
	st_ctrl_out					: struct_ctrl_out;
	haspel1_ctrl_out				: struct_ctrl_in;
	haspel2_ctrl_out				: struct_ctrl_in;
	b_materialmangel_bandende	: BOOL := FALSE;
END_VAR
VAR
	fb_ton_wz					: TON;
	fb_ton_uez					: TON;
	fb_ton_vz					: TON;
	fb_tof_motor					: TOF;
	fb_ton_quitt					: TON;
	fb_r_trig_start					: R_TRIG;
	fb_state_entry					: ST_StateEntry;
	sm_haspel_nicht_bb			: BOOL := FALSE;
	e_haspelmotor_bb			AT %I* : BOOL;
	a_motor_drehrichtung_rechts	AT %Q* : BOOL;
	a_motor_drehrichtung_links		AT %Q* : BOOL;
END_VAR
(* Zeiten *)
fb_ton_wz(IN:= , PT:= , Q=>  , ET=> );
fb_ton_uez(IN:= , PT:= , Q=>  , ET=> );
fb_ton_vz(IN:= , PT:= , Q=>  , ET=> );
fb_tof_motor(IN:= , PT:= t_abschaltzeit_motor, Q=> , ET=> );
fb_ton_quitt(IN:= , PT:= t#100ms, Q=> , ET=> );

(* Flanken *)
fb_r_trig_start(CLK:= st_ctrl_in.b_start, Q=> );

(* Haspelmotor *)
IF 	e_steuerung_ein AND
	e_druckwaechter AND
	fb_tof_motor.Q AND
	fb_state_entry.i16_next_step <> FEHLER THEN
		a_motor_drehrichtung_links 	:= b_drehrichtung_antrieb_links;
		a_motor_drehrichtung_rechts := NOT b_drehrichtung_antrieb_links;
ELSE
	a_motor_drehrichtung_links 	:= FALSE;
	a_motor_drehrichtung_rechts := FALSE;
END_IF

(* Freigabe für die jeweils benutzte Haspel setzen. Wird für Bandende benötigt (ST_Haspel_V2)*)
CASE gst_datensatz.st_md.i16_typ_zelle OF

KEINE_ZELLE:
		;

BESTUECKZELLE_1700:
	IF zyl_bandeinzuege_verschieben.st_ctrl.out.b_ausgefahren THEN
		haspel1_ctrl_out.b_freigabe := TRUE;
		haspel2_ctrl_out.b_freigabe := FALSE;
	ELSIF zyl_bandeinzuege_verschieben.st_ctrl.out.b_eingefahren THEN
		haspel1_ctrl_out.b_freigabe := FALSE;
		haspel2_ctrl_out.b_freigabe := TRUE;
	END_IF

RASTERFOLIE:
	haspel1_ctrl_out.b_freigabe := TRUE;
	haspel2_ctrl_out.b_freigabe := FALSE;

BESTUECKZELLE_1720:
	haspel1_ctrl_out.b_freigabe := TRUE;
	haspel2_ctrl_out.b_freigabe := TRUE;

END_CASE

(* Bandende von Haspel rechts bzw. links *)
IF	(gi16_betriebsart = AUTO OR gi16_betriebsart = TIPPEN) AND
	(haspel1_ctrl_in.b_bandende OR haspel2_ctrl_in.b_bandende )
	THEN
		st_ctrl_out.b_bandende := b_materialmangel_bandende := TRUE;
ELSE
		st_ctrl_out.b_bandende := b_materialmangel_bandende := FALSE;
END_IF

(* Toplevel *)
IF fb_state_entry.i16_next_step > INIT AND fb_state_entry.i16_next_step < FEHLER THEN
	IF fb_state_entry.i16_next_step < STOP THEN
		IF st_ctrl_in.b_stop THEN
			fb_state_entry.i16_next_step := STOP;
		END_IF
	END_IF
	(* Allgemeine Fehler *)
	IF haspel1_ctrl_in.b_fehler OR haspel2_ctrl_in.b_fehler THEN
		fb_state_entry.i16_next_step := FEHLER;
	END_IF
END_IF


(* ======================================Schrittkette======================================== *)
fb_state_entry(
	i16_next_step:= ,
	i16_pos:= 1,
	s_debugtext:= ,
	E=> ,
	X=> , 
	i16_step=> ,
	i16_last_step=> );

CASE fb_state_entry.i16_step OF
(*=======================================================*)
	INIT_OBJ:
		IF st_config.b_config_fertig THEN
			fb_state_entry.i16_next_step := INIT;
		END_IF

(*=======================================================*)
	INIT:
		IF fb_state_entry.E THEN
			fb_ton_wz.IN := FALSE;
			fb_ton_uez.IN	:= FALSE;
			fb_ton_vz.IN := FALSE;
			fb_ton_quitt.IN := FALSE;
			a_motor_drehrichtung_links := FALSE;
			a_motor_drehrichtung_rechts := FALSE;
			sm_haspel_nicht_bb := FALSE;
			st_ctrl_out.b_fehler := FALSE;
			st_ctrl_out.b_bereit := FALSE;
			st_ctrl_out.b_fertig := FALSE;
			haspel1_ctrl_out.b_stop := FALSE;
			haspel2_ctrl_out.b_stop := FALSE;
			haspel1_ctrl_out.b_init := FALSE;
			haspel2_ctrl_out.b_init := FALSE;
		END_IF

		(*-----------------------Weiterschaltbedingungen----------------------------*)
		IF st_ctrl_in.b_init THEN
			haspel1_ctrl_out.b_quitt := FALSE;
			haspel2_ctrl_out.b_quitt := FALSE;
			fb_state_entry.i16_next_step :=20;
		END_IF

(*=======================================================*)
	20:	(* Haspeln initialisieren *)
		IF fb_state_entry.E THEN
			haspel1_ctrl_out.b_init := TRUE;
			haspel2_ctrl_out.b_init := TRUE;
		END_IF

		(*-----------------------Weiterschaltbedingungen----------------------------*)
		IF  haspel1_ctrl_in.b_bereit AND haspel2_ctrl_in.b_bereit THEN
			haspel1_ctrl_out.b_init := FALSE;
			haspel2_ctrl_out.b_init := FALSE;
			fb_tof_motor.IN := TRUE;
			fb_state_entry.i16_next_step := BEREIT;
		END_IF

(*=======================================================*)
	BEREIT: (* Haspelmotor läuft *)
		IF fb_state_entry.E THEN
			st_ctrl_out.b_bereit := TRUE;
			st_ctrl_out.b_fertig := TRUE;
		END_IF

		IF haspel1_ctrl_in.b_kontroller_start OR haspel2_ctrl_in.b_kontroller_start THEN	(* Abschaltzeit für Haspelmotor nachtriggern*)
			fb_tof_motor.IN := TRUE;
		ELSE
			fb_tof_motor.IN := FALSE;
		END_IF

(*=======================================================*)
	FEHLER:
		IF fb_state_entry.E THEN
			st_ctrl_out.b_fehler := TRUE;
			fb_tof_motor.IN := FALSE;
			haspel1_ctrl_out.b_quitt := FALSE;
			haspel2_ctrl_out.b_quitt := FALSE;
			haspel1_ctrl_out.b_stop := FALSE;
			haspel2_ctrl_out.b_stop := FALSE;
			fb_ton_quitt.IN := FALSE;
		END_IF

		(*-----------------------Weiterschaltbedingungen----------------------------*)
		IF st_ctrl_in.b_quitt AND NOT fb_state_entry.E THEN
			haspel1_ctrl_out.b_quitt := TRUE;
			haspel2_ctrl_out.b_quitt := TRUE;
			st_ctrl_out.b_fehler := FALSE;
			fb_ton_quitt.IN := TRUE;
		END_IF

		IF fb_ton_quitt.Q THEN
			fb_ton_quitt.IN := FALSE;
			fb_state_entry.i16_next_step := INIT;
		END_IF

(*=======================================================*)
	STOP:
		IF fb_state_entry.E THEN
			fb_tof_motor.IN := FALSE;
			haspel1_ctrl_out.b_stop := TRUE;
			haspel2_ctrl_out.b_stop := TRUE;
			haspel1_ctrl_out.b_quitt := FALSE;
			haspel2_ctrl_out.b_quitt := FALSE;
			fb_ton_quitt.IN := FALSE;
		END_IF

		(*-----------------------Weiterschaltbedingungen----------------------------*)
		IF st_ctrl_in.b_quitt AND NOT fb_state_entry.E THEN
			haspel1_ctrl_out.b_stop := FALSE;
			haspel2_ctrl_out.b_stop := FALSE;
			haspel1_ctrl_out.b_quitt := TRUE;
			haspel2_ctrl_out.b_quitt := TRUE;
			fb_ton_quitt.IN := TRUE;
		END_IF

		IF fb_ton_quitt.Q THEN
			fb_ton_quitt.IN := FALSE;
			fb_state_entry.i16_next_step := INIT;
		END_IF
END_CASE

fb_state_entry(
	i16_next_step:= , 
	i16_pos:= 2,
	s_debugtext:= ,
	E=> , 
	X=> , 
	i16_step=> ,
	i16_last_step=> );

IF st_config.b_config_fertig THEN
	(* Fehlermeldungen und Betriebsmeldungen ab dem Startindex in die globalen Meldungsarrays schreiben *)
	garr_stoermeldungen[st_config.i16_meld_startindex + 0] := sm_haspel_nicht_bb;
	garr_stoermeldungen[st_config.i16_meld_startindex + 1] := FALSE;
	garr_stoermeldungen[st_config.i16_meld_startindex + 2] := FALSE;
	garr_stoermeldungen[st_config.i16_meld_startindex + 3] := FALSE;
	garr_stoermeldungen[st_config.i16_meld_startindex + 4] := FALSE;
	garr_stoermeldungen[st_config.i16_meld_startindex + 5] := FALSE;
	garr_stoermeldungen[st_config.i16_meld_startindex + 6] := FALSE;
	garr_stoermeldungen[st_config.i16_meld_startindex + 7] := FALSE;
	garr_stoermeldungen[st_config.i16_meld_startindex + 8] := FALSE;
	garr_stoermeldungen[st_config.i16_meld_startindex + 9] := FALSE;
	garr_stoermeldungen[st_config.i16_meld_startindex + 10] := FALSE;
	garr_stoermeldungen[st_config.i16_meld_startindex + 11] := FALSE;
	garr_stoermeldungen[st_config.i16_meld_startindex + 12] := FALSE;
	garr_stoermeldungen[st_config.i16_meld_startindex + 13] := FALSE;
	garr_stoermeldungen[st_config.i16_meld_startindex + 14] := FALSE;
	garr_stoermeldungen[st_config.i16_meld_startindex + 15] := FALSE;
	garr_stoermeldungen[st_config.i16_meld_startindex + 16] := FALSE;
	garr_stoermeldungen[st_config.i16_meld_startindex + 17] := FALSE;
	garr_stoermeldungen[st_config.i16_meld_startindex + 18] := FALSE;
	garr_stoermeldungen[st_config.i16_meld_startindex + 19] := FALSE;
	
	garr_betriebsmeldungen[st_config.i16_meld_startindex + 0] := FALSE;
	garr_betriebsmeldungen[st_config.i16_meld_startindex + 1] := FALSE;
	garr_betriebsmeldungen[st_config.i16_meld_startindex + 2] := FALSE;
	garr_betriebsmeldungen[st_config.i16_meld_startindex + 3] := FALSE;
	garr_betriebsmeldungen[st_config.i16_meld_startindex + 4] := FALSE;
	garr_betriebsmeldungen[st_config.i16_meld_startindex + 5] := FALSE;
	garr_betriebsmeldungen[st_config.i16_meld_startindex + 6] := FALSE;
	garr_betriebsmeldungen[st_config.i16_meld_startindex + 7] := FALSE;
	garr_betriebsmeldungen[st_config.i16_meld_startindex + 8] := FALSE;
	garr_betriebsmeldungen[st_config.i16_meld_startindex + 9] := FALSE;
	garr_betriebsmeldungen[st_config.i16_meld_startindex + 10] := FALSE;
	garr_betriebsmeldungen[st_config.i16_meld_startindex + 11] := FALSE;
	garr_betriebsmeldungen[st_config.i16_meld_startindex + 12] := FALSE;
	garr_betriebsmeldungen[st_config.i16_meld_startindex + 13] := FALSE;
	garr_betriebsmeldungen[st_config.i16_meld_startindex + 14] := FALSE;
	garr_betriebsmeldungen[st_config.i16_meld_startindex + 15] := FALSE;
	garr_betriebsmeldungen[st_config.i16_meld_startindex + 16] := FALSE;
	garr_betriebsmeldungen[st_config.i16_meld_startindex + 17] := FALSE;
	garr_betriebsmeldungen[st_config.i16_meld_startindex + 18] := FALSE;
	garr_betriebsmeldungen[st_config.i16_meld_startindex + 19] := FALSE;
END_IF
END_PROGRAM

(* POU Gemeinsamkeiten17xx/Oeler/ST_Menzel_Spruehoeler, ST *)
PROGRAM ST_Menzel_Spruehoeler
VAR_INPUT
	st_config						: struct_config;
	st_ctrl_in						: struct_ctrl_in;
	lr_achse_position				: LREAL;
	e_steuerung_ein				: BOOL;
	e_druckwaechter				: BOOL;
END_VAR
(*VAR_IN_OUT
	st_visu						: struct_oeler_visu;
END_VAR*)
VAR_OUTPUT
	st_ctrl_out					: struct_ctrl_out;
	b_oelmangel					: BOOL;
END_VAR
VAR
	fb_ton_uez					: TON;
	fb_ton_uez_fuellstand			: TON;
	fb_ton_quitt					: TON;
	fb_ton_speichern			: TON;
	fb_state_entry				: ST_StateEntry;
	fb_winkeltrigger				: ST_Winkeltrigger;
	b_hand_dialog_aktiv			: BOOL := FALSE;
	a_ventil			 			AT %Q* : BOOL;
	e_fuellstand					AT %I* : BOOL;
	e_druck_oelbehaelter			AT %I* : BOOL;
	sm_fuellstand_oeler			: BOOL := FALSE;
	sm_druckueberwachung		: BOOL := FALSE;
	bm_fuellstand_oeler			: BOOL := FALSE;
	b_ibn_handoelen				: BOOL := FALSE;
	fb_betriebsartenwechsel		: ST_Betriebsartenwechsel;
	fb_r_trig_bestueckhub			: R_TRIG;
	i16_hubzaehler				: INT := 0;
	fb_ton_oelen					: TON;
END_VAR
(*Intervalllölen wird beim Sprühöler nicht mehr benötigt, darum wird der Wert auf Null geforced*)
gst_datensatz.st_wkz.st_oeler.i16_intervall_bandoelen:=0;

(*Mindestwerte eintragen damit nicht trocken gefahren werden kann*)
fb_ton_speichern(IN:= gst_datensatz.st_wkz.st_oeler.t_ventiloeffnungszeit<500 OR gst_datensatz.st_wkz.st_oeler.i16_intervall_bandoelen<1, PT:= t#20ms, Q=> , ET=> );
IF	fb_ton_speichern.Q THEN
	IF	gst_datensatz.st_wkz.st_oeler.t_ventiloeffnungszeit<500 THEN
		gst_datensatz.st_wkz.st_oeler.t_ventiloeffnungszeit:=500;
	END_IF

	IF	gst_datensatz.st_wkz.st_oeler.i16_intervall_bandoelen<1 THEN
		gst_datensatz.st_wkz.st_oeler.i16_intervall_bandoelen:=0;
	END_IF
END_IF

(* Bandöler mit Füllstandsabfrage *)
fb_ton_quitt(IN:= , PT:= t#100ms, Q=> , ET=> );
fb_ton_uez(IN:= NOT e_druck_oelbehaelter AND e_druckwaechter, PT:= t#60s, Q=> , ET=> );
fb_ton_uez_fuellstand(IN:= bm_fuellstand_oeler, PT:= t#1h, Q=> , ET=> );
fb_ton_oelen(IN:= , PT:= , Q=> , ET=> );

IF fb_state_entry.i16_step >= BEREIT AND fb_state_entry.i16_step < FEHLER THEN
	fb_winkeltrigger(IN:= LREAL_TO_INT(lr_achse_position), PT:= T#300ms, Q=> );
END_IF

(* Flanken *)
fb_r_trig_bestueckhub(CLK:= (gi16_betriebsart = AUTO OR gi16_betriebsart = TIPPEN) AND nockenschaltwerk_bestueckachse.fb.arr_spur[SP_OT], Q=> );

(* Hubzähler wird durch Nocke OT erhöht >> wenn der Zähler größer gleich dem Intervall ist wird a_ventil gesetzt *)
IF fb_r_trig_bestueckhub.Q THEN
	i16_hubzaehler := i16_hubzaehler + 1;
END_IF

(* Bandöler von Hand betätigen *)
IF gi16_betriebsart = HAND THEN
	a_ventil :=  b_ibn_handoelen OR (b_hand_dialog_aktiv AND (visu.b_handoelen OR ST_Euchner_Handbedienpult.b_Taste_Power));
END_IF

fb_betriebsartenwechsel(
	i16_akt_betriebsart:= gi16_betriebsart,
	b_wechsel_auto=> , 
	b_wechsel_tippen=> ,
	b_wechsel_hand=> , 
	b_wechsel_dummy=> , 
	b_wechsel_pseudo=> , 
	b_wechsel_allgemein=> );
(*
IF fb_betriebsartenwechsel.b_merker_ba_auto OR fb_betriebsartenwechsel.b_merker_ba_tippen THEN
	a_ventil := FALSE;
END_IF
*)

(* =======================================Toplevel========================================== *)
IF fb_state_entry.i16_next_step > INIT AND fb_state_entry.i16_next_step < FEHLER THEN
	IF fb_state_entry.i16_next_step < STOP THEN
		IF st_ctrl_in.b_stop THEN
			fb_state_entry.i16_next_step := STOP;
		END_IF
	END_IF
END_IF

(* Orangene Lampe an Ampel leuchtet bei Ölbehälter leer *)
b_oelmangel := bm_fuellstand_oeler;

(* ==================================Schrittkette================================ *)
fb_state_entry(
	i16_next_step:= , 
	i16_pos:= 1,
	s_debugtext:= ,
	E=> ,
	X=> ,
	i16_step=> ,
	i16_last_step=> );

CASE fb_state_entry.i16_step OF
(*=======================================================*)
	INIT_OBJ:
		IF st_config.b_config_fertig THEN
			fb_state_entry.i16_next_step := INIT;
		END_IF
		
(*=======================================================*)
	INIT:
		IF fb_state_entry.E THEN
			st_ctrl_out.b_fehler := FALSE;
			st_ctrl_out.b_bereit := FALSE;
			st_ctrl_out.b_fertig := FALSE;
			fb_ton_quitt.IN := FALSE;
			fb_ton_uez_fuellstand.IN := FALSE;
			a_ventil := FALSE;
			sm_fuellstand_oeler := FALSE;
			sm_druckueberwachung := FALSE;
			bm_fuellstand_oeler := FALSE;
			st_ctrl_out.b_einzelfertigung := FALSE;
			fb_ton_oelen.IN := FALSE;
		END_IF

		(*-----------------------Weiterschaltbedingungen----------------------------*)
		IF st_ctrl_in.b_init THEN
			fb_state_entry.i16_next_step := BEREIT;
		END_IF

(*=======================================================*)
	BEREIT:
		IF fb_state_entry.E THEN
			st_ctrl_out.b_bereit := TRUE;
		END_IF

		IF st_config.b_station_aktiv THEN
			(* Ölen *)
			IF (gi16_betriebsart = AUTO OR gi16_betriebsart = TIPPEN) THEN
				IF	gst_datensatz.st_wkz.st_oeler.i16_intervall_bandoelen =0 THEN  (*bei Intervall 0 Dauerölen*)
					a_ventil :=  fb_winkeltrigger.Q OR visu.b_handoelen OR b_ibn_handoelen;
				ELSE
					a_ventil :=  visu.b_handoelen OR b_ibn_handoelen;
				END_IF
			END_IF
			(* Überwachung Füllstand Betriebsmeldung*)
			IF NOT e_fuellstand AND e_steuerung_ein THEN
				bm_fuellstand_oeler := TRUE;
			ELSE
				bm_fuellstand_oeler := FALSE;
			END_IF
			(* Überwachung Füllstand Störmeldung *)
			IF fb_ton_uez_fuellstand.Q OR sm_fuellstand_oeler THEN
				sm_fuellstand_oeler := TRUE;
				st_ctrl_out.b_einzelfertigung:=TRUE;

				IF 	gi16_maschinenstatusinfo = STATUS_BETRIEBSBEREIT THEN
					fb_state_entry.i16_next_step := FEHLER;
				END_IF

			END_IF
			(* Überwachung Druck im Ölbehälter *)
			IF fb_ton_uez.Q OR sm_druckueberwachung THEN
				sm_druckueberwachung := TRUE;
				st_ctrl_out.b_einzelfertigung:=TRUE;

				IF 	gi16_maschinenstatusinfo = STATUS_BETRIEBSBEREIT THEN
					fb_state_entry.i16_next_step := FEHLER;
				END_IF
			END_IF

			(*-----------------------Weiterschaltbedingungen----------------------------*)
			IF	 i16_hubzaehler >= gst_datensatz.st_wkz.st_oeler.i16_intervall_bandoelen AND
				gst_datensatz.st_wkz.st_oeler.i16_intervall_bandoelen <>0 THEN (*bei Intervall 0 Dauerölen*)
				fb_state_entry.i16_next_step := 110;
			END_IF

		END_IF

(*=======================================================*)
	110: (* Bandölen, abhängig von WKZ-Daten *)
		IF fb_state_entry.E THEN
			i16_hubzaehler := 0;
			fb_ton_oelen.IN := TRUE;
			fb_ton_oelen.PT := DINT_TO_TIME(gst_datensatz.st_wkz.st_oeler.t_ventiloeffnungszeit);
			a_ventil := TRUE;
		END_IF

		(*-----------------------Weiterschaltbedingungen----------------------------*)
		IF fb_ton_oelen.Q THEN
			fb_ton_oelen.IN := FALSE;
			a_ventil := FALSE;
			fb_state_entry.i16_next_step := BEREIT;
		END_IF

(*=======================================================*)
	FEHLER:
		IF fb_state_entry.E THEN
			st_ctrl_out.b_fehler := TRUE;
			a_ventil := FALSE;
			fb_ton_quitt.IN := FALSE;
		END_IF

		(*-----------------------Weiterschaltbedingungen----------------------------*)
		IF st_ctrl_in.b_quitt AND NOT fb_state_entry.E THEN
			st_ctrl_out.b_fehler := FALSE;
			fb_ton_quitt.IN := TRUE;
		END_IF

		IF fb_ton_quitt.Q THEN
			fb_ton_quitt.IN := FALSE;
			fb_state_entry.i16_next_step := INIT;
		END_IF

(*=======================================================*)
	STOP:
		IF fb_state_entry.E THEN
			a_ventil := FALSE;
			fb_ton_quitt.IN := FALSE;
		END_IF

		(*-----------------------Weiterschaltbedingungen----------------------------*)
		IF st_ctrl_in.b_quitt AND NOT fb_state_entry.E THEN
			fb_ton_quitt.IN := TRUE;
		END_IF

		IF fb_ton_quitt.Q THEN
			fb_ton_quitt.IN := FALSE;
			fb_state_entry.i16_next_step := INIT;
		END_IF
END_CASE

fb_state_entry(
	i16_next_step:= , 
	i16_pos:= 2,
	s_debugtext:= ,
	E=> ,
	X=> , 
	i16_step=> ,
	i16_last_step=> );

IF st_config.b_config_fertig THEN
	(* Fehlermeldungen und Betriebsmeldungen ab dem Startindex in die globalen Meldungsarrays schreiben *)
	garr_stoermeldungen[st_config.i16_meld_startindex + 0] := sm_fuellstand_oeler;
	garr_stoermeldungen[st_config.i16_meld_startindex + 1] := sm_druckueberwachung;
	garr_stoermeldungen[st_config.i16_meld_startindex + 2] := FALSE;
	garr_stoermeldungen[st_config.i16_meld_startindex + 3] := FALSE;
	garr_stoermeldungen[st_config.i16_meld_startindex + 4] := FALSE;
	garr_stoermeldungen[st_config.i16_meld_startindex + 5] := FALSE;
	garr_stoermeldungen[st_config.i16_meld_startindex + 6] := FALSE;
	garr_stoermeldungen[st_config.i16_meld_startindex + 7] := FALSE;
	garr_stoermeldungen[st_config.i16_meld_startindex + 8] := FALSE;
	garr_stoermeldungen[st_config.i16_meld_startindex + 9] := FALSE;
	garr_stoermeldungen[st_config.i16_meld_startindex + 10] := FALSE;
	garr_stoermeldungen[st_config.i16_meld_startindex + 11] := FALSE;
	garr_stoermeldungen[st_config.i16_meld_startindex + 12] := FALSE;
	garr_stoermeldungen[st_config.i16_meld_startindex + 13] := FALSE;
	garr_stoermeldungen[st_config.i16_meld_startindex + 14] := FALSE;
	garr_stoermeldungen[st_config.i16_meld_startindex + 15] := FALSE;
	garr_stoermeldungen[st_config.i16_meld_startindex + 16] := FALSE;
	garr_stoermeldungen[st_config.i16_meld_startindex + 17] := FALSE;
	garr_stoermeldungen[st_config.i16_meld_startindex + 18] := FALSE;
	garr_stoermeldungen[st_config.i16_meld_startindex + 19] := FALSE;
	
	garr_betriebsmeldungen[st_config.i16_meld_startindex + 0] := bm_fuellstand_oeler;
	garr_betriebsmeldungen[st_config.i16_meld_startindex + 1] := FALSE;
	garr_betriebsmeldungen[st_config.i16_meld_startindex + 2] := FALSE;
	garr_betriebsmeldungen[st_config.i16_meld_startindex + 3] := FALSE;
	garr_betriebsmeldungen[st_config.i16_meld_startindex + 4] := FALSE;
	garr_betriebsmeldungen[st_config.i16_meld_startindex + 5] := FALSE;
	garr_betriebsmeldungen[st_config.i16_meld_startindex + 6] := FALSE;
	garr_betriebsmeldungen[st_config.i16_meld_startindex + 7] := FALSE;
	garr_betriebsmeldungen[st_config.i16_meld_startindex + 8] := FALSE;
	garr_betriebsmeldungen[st_config.i16_meld_startindex + 9] := FALSE;
	garr_betriebsmeldungen[st_config.i16_meld_startindex + 10] := FALSE;
	garr_betriebsmeldungen[st_config.i16_meld_startindex + 11] := FALSE;
	garr_betriebsmeldungen[st_config.i16_meld_startindex + 12] := FALSE;
	garr_betriebsmeldungen[st_config.i16_meld_startindex + 13] := FALSE;
	garr_betriebsmeldungen[st_config.i16_meld_startindex + 14] := FALSE;
	garr_betriebsmeldungen[st_config.i16_meld_startindex + 15] := FALSE;
	garr_betriebsmeldungen[st_config.i16_meld_startindex + 16] := FALSE;
	garr_betriebsmeldungen[st_config.i16_meld_startindex + 17] := FALSE;
	garr_betriebsmeldungen[st_config.i16_meld_startindex + 18] := FALSE;
	garr_betriebsmeldungen[st_config.i16_meld_startindex + 19] := FALSE;
END_IF
END_PROGRAM

(* POU EPT Lib/Funktionsbausteine/ST_Winkeltrigger, ST *)
FUNCTION_BLOCK ST_Winkeltrigger
VAR_INPUT
	IN							: DINT;
	PT							: TIME;
END_VAR
VAR_OUTPUT
	Q							: BOOL;
END_VAR
VAR
	i32_alter_winkel				: DINT := 0;
	i32_neuer_winkel				: DINT := 0;
	b_triggersignal_start			: BOOL := FALSE;
	fb_tof_triggersignal			: TOF;
	t_zeit						: TIME := t#0ms;
END_VAR
(* Sobald sich der Hauptantrieb dreht, wird ein Triggersignal von mindestens 200ms erzeugt um Aktionen auszulösen *)
i32_neuer_winkel := IN;

IF PT < t#200ms THEN
	t_zeit := t#200ms;
ELSE
	t_zeit := PT;
END_IF

IF i32_neuer_winkel <> 360 THEN
	IF i32_neuer_winkel > i32_alter_winkel OR i32_neuer_winkel < i32_alter_winkel THEN
		b_triggersignal_start := TRUE;
	ELSE
		b_triggersignal_start := FALSE;
	END_IF
	i32_alter_winkel := i32_neuer_winkel;
ELSE
	b_triggersignal_start := FALSE;
END_IF

fb_tof_triggersignal(IN:= b_triggersignal_start, PT:= t_zeit, Q=> Q, ET=> );
END_FUNCTION_BLOCK

(* POU EPT Lib/Funktionsbausteine/ST_Betriebsartenwechsel, ST *)
FUNCTION_BLOCK ST_Betriebsartenwechsel
VAR_INPUT
	i16_akt_betriebsart		: enum_betriebsarten;
END_VAR
VAR_OUTPUT
	b_wechsel_auto			: BOOL;
	b_wechsel_tippen			: BOOL;
	b_wechsel_hand			: BOOL;
	b_wechsel_dummy		: BOOL;
	b_wechsel_pseudo		: BOOL;
	b_wechsel_allgemein		: BOOL;
END_VAR
VAR
	fb_r_trig_ba_auto			: R_TRIG;
	fb_r_trig_ba_tippen		: R_TRIG;
	fb_r_trig_ba_hand			: R_TRIG;
	fb_r_trig_ba_dummy		: R_TRIG;
	fb_r_trig_ba_pseudo		: R_TRIG;
	i16_betriebsart_alt			: enum_betriebsarten := KEINE;
	i16_betriebsart_neu		: enum_betriebsarten := KEINE;
	b_merker_ba_auto		: BOOL := FALSE;
	b_merker_ba_tippen		: BOOL := FALSE;
	b_merker_ba_hand		: BOOL := FALSE;
	b_merker_ba_dummy		: BOOL := FALSE;
	b_merker_ba_pseudo		: BOOL := FALSE;
END_VAR
(* Funktionsbaustein zum Erfassen der verschiedenen Betriebsartenflanken *)
fb_r_trig_ba_auto(CLK:= b_merker_ba_auto, Q=> b_wechsel_auto);
fb_r_trig_ba_tippen(CLK:= b_merker_ba_tippen, Q=> b_wechsel_tippen);
fb_r_trig_ba_hand(CLK:=b_merker_ba_hand , Q=> b_wechsel_hand);
fb_r_trig_ba_dummy(CLK:=b_merker_ba_dummy , Q=> b_wechsel_dummy);
fb_r_trig_ba_pseudo(CLK:=b_merker_ba_pseudo , Q=> b_wechsel_pseudo);

b_wechsel_allgemein := b_wechsel_auto OR b_wechsel_tippen OR b_wechsel_hand OR b_wechsel_dummy OR b_wechsel_pseudo;

i16_betriebsart_neu := i16_akt_betriebsart;

IF i16_betriebsart_neu <> i16_betriebsart_alt THEN
	CASE gi16_betriebsart OF
		KEINE:
			b_merker_ba_auto := FALSE;
			b_merker_ba_tippen := FALSE;
			b_merker_ba_hand := FALSE;
			b_merker_ba_dummy := FALSE;
			b_merker_ba_pseudo := FALSE;

		AUTO:
			b_merker_ba_auto := TRUE;
			b_merker_ba_tippen := FALSE;
			b_merker_ba_hand := FALSE;
			b_merker_ba_dummy := FALSE;
			b_merker_ba_pseudo := FALSE;

		TIPPEN:
			b_merker_ba_auto := FALSE;
			b_merker_ba_tippen := TRUE;
			b_merker_ba_hand := FALSE;
			b_merker_ba_dummy := FALSE;
			b_merker_ba_pseudo := FALSE;

		HAND:
			b_merker_ba_auto := FALSE;
			b_merker_ba_tippen := FALSE;
			b_merker_ba_hand := TRUE;
			b_merker_ba_dummy := FALSE;
			b_merker_ba_pseudo := FALSE;

		DUMMY:
			b_merker_ba_auto := FALSE;
			b_merker_ba_tippen := FALSE;
			b_merker_ba_hand := FALSE;
			b_merker_ba_dummy := TRUE;
			b_merker_ba_pseudo := FALSE;

		PSEUDO:
			b_merker_ba_auto := FALSE;
			b_merker_ba_tippen := FALSE;
			b_merker_ba_hand := FALSE;
			b_merker_ba_dummy := FALSE;
			b_merker_ba_pseudo := TRUE;
	END_CASE

	i16_betriebsart_alt := i16_betriebsart_neu;
END_IF
END_FUNCTION_BLOCK

(* POU Gemeinsamkeiten17xx/Oeler/ST_BandoelerZylinder, ST *)
PROGRAM ST_BandoelerZylinder
VAR_INPUT
	st_config						: struct_config;
	st_ctrl_in						: struct_ctrl_in;
	lr_achse_position				: LREAL;
	e_steuerung_ein				: BOOL;
	e_druckwaechter				: BOOL;

END_VAR
(*VAR_IN_OUT
	st_visu						: struct_oeler_visu;
END_VAR*)
VAR_OUTPUT
	st_ctrl_out					: struct_ctrl_out;
	b_oelmangel					: BOOL;
	st_oelerdaten					: struct_oeler_daten;
END_VAR
VAR
	fb_ton_uez					: TON;
	fb_ton_uez_fuellstand			: TON;
	fb_ton_quitt					: TON;
	fb_ton_speichern			: TON;
	fb_state_entry				: ST_StateEntry;
	fb_winkeltrigger				: ST_Winkeltrigger;
	b_hand_dialog_aktiv			: BOOL := FALSE;
	a_ventil_oben			 			AT %Q* : BOOL;
	a_ventil_unten			 			AT %Q* : BOOL;
	e_fuellstand					AT %I* : BOOL;
	e_druck_oelbehaelter			AT %I* : BOOL;
	sm_fuellstand_oeler			: BOOL := FALSE;
	sm_druckueberwachung		: BOOL := FALSE;
	bm_fuellstand_oeler			: BOOL := FALSE;
	b_ibn_handoelen				: BOOL := FALSE;
	fb_betriebsartenwechsel		: ST_Betriebsartenwechsel;
	fb_r_trig_bestueckhub			: R_TRIG;
	i16_hubzaehler				: INT := 0;
	fb_ton_oelen					: TON;
	b_zyl_unten					: BOOL;
	b_zyl_oben					: BOOL;
	dt_datum_uhrzeit_letzte_oelung	: DT;
	t_delta_zeitraum				: TIME := t#5h;
	fb_ton_oelzeit					: TON;
END_VAR
(*Mindestwerte eintragen damit nicht trocken gefahren werden kann*)
fb_ton_speichern(IN:= gst_datensatz.st_wkz.st_oeler.t_ventiloeffnungszeit<500 OR gst_datensatz.st_wkz.st_oeler.i16_intervall_bandoelen<1, PT:= t#20ms, Q=> , ET=> );
IF	fb_ton_speichern.Q THEN
	IF	gst_datensatz.st_wkz.st_oeler.t_ventiloeffnungszeit<50 THEN
		gst_datensatz.st_wkz.st_oeler.t_ventiloeffnungszeit:=500;
	END_IF

	IF	gst_datensatz.st_wkz.st_oeler.i16_intervall_bandoelen<1 THEN
		gst_datensatz.st_wkz.st_oeler.i16_intervall_bandoelen:=0;
	END_IF
END_IF

(* Bandöler mit Füllstandsabfrage *)
fb_ton_quitt(IN:= , PT:= t#100ms, Q=> , ET=> );
fb_ton_uez(IN:= NOT e_druck_oelbehaelter AND e_druckwaechter, PT:= t#60s, Q=> , ET=> );
fb_ton_uez_fuellstand(IN:= bm_fuellstand_oeler, PT:= t#1h, Q=> , ET=> );
fb_ton_oelen(IN:= , PT:= , Q=> , ET=> );

IF fb_state_entry.i16_step >= BEREIT AND fb_state_entry.i16_step < FEHLER THEN
	fb_winkeltrigger(IN:= LREAL_TO_INT(lr_achse_position), PT:= T#300ms, Q=> );
END_IF

(* Flanken *)
fb_r_trig_bestueckhub(CLK:= (gi16_betriebsart = AUTO OR gi16_betriebsart = TIPPEN) AND nockenschaltwerk_bestueckachse.fb.arr_spur[SP_OT], Q=> );

(* Hubzähler wird durch Nocke OT erhöht >> wenn der Zähler größer gleich dem Intervall ist wird a_ventil gesetzt *)
IF fb_r_trig_bestueckhub.Q THEN
	i16_hubzaehler := i16_hubzaehler + 1;
END_IF


(* Bandöler von Hand betätigen *)
IF gi16_betriebsart = HAND THEN
	a_ventil_oben :=  b_ibn_handoelen OR visu.b_handoelen ;
	a_ventil_unten :=  b_ibn_handoelen OR visu.b_handoelen ;
END_IF


(* Allgemeine Fehler *)

IF zyl_oelen_unten.st_ctrl.out.b_fehler OR
	zyl_oelen_oben.st_ctrl.out.b_fehler THEN
	fb_state_entry.i16_next_step := FEHLER;
END_IF

fb_betriebsartenwechsel(
	i16_akt_betriebsart:= gi16_betriebsart,
	b_wechsel_auto=> , 
	b_wechsel_tippen=> ,
	b_wechsel_hand=> , 
	b_wechsel_dummy=> , 
	b_wechsel_pseudo=> , 
	b_wechsel_allgemein=> );
(*
IF fb_betriebsartenwechsel.b_merker_ba_auto OR fb_betriebsartenwechsel.b_merker_ba_tippen THEN
	a_ventil := FALSE;
END_IF
*)

(* =======================================Toplevel========================================== *)
IF fb_state_entry.i16_next_step > INIT AND fb_state_entry.i16_next_step < FEHLER THEN
	IF fb_state_entry.i16_next_step < STOP THEN
		IF st_ctrl_in.b_stop THEN
			fb_state_entry.i16_next_step := STOP;
		END_IF
	END_IF
END_IF

(* Orangene Lampe an Ampel leuchtet bei Ölbehälter leer *)
b_oelmangel := bm_fuellstand_oeler;

(* ==================================Schrittkette================================ *)
fb_state_entry(
	i16_next_step:= , 
	i16_pos:= 1,
	s_debugtext:= ,
	E=> ,
	X=> ,
	i16_step=> ,
	i16_last_step=> );

CASE fb_state_entry.i16_step OF
(*=======================================================*)
	INIT_OBJ:
		IF st_config.b_config_fertig THEN
			fb_state_entry.i16_next_step := INIT;
		END_IF
		
(*=======================================================*)
	INIT:
		IF fb_state_entry.E THEN
			st_ctrl_out.b_fehler := FALSE;
			st_ctrl_out.b_bereit := FALSE;
			st_ctrl_out.b_fertig := FALSE;
			fb_ton_quitt.IN := FALSE;
			fb_ton_uez_fuellstand.IN := FALSE;
			a_ventil_oben := FALSE;
			a_ventil_unten := FALSE;
			sm_fuellstand_oeler := FALSE;
			sm_druckueberwachung := FALSE;
			bm_fuellstand_oeler := FALSE;
			st_ctrl_out.b_einzelfertigung := FALSE;
			fb_ton_oelen.IN := FALSE;
			b_zyl_unten:= FALSE;
			b_zyl_oben:= FALSE;
		END_IF

		(*-----------------------Weiterschaltbedingungen----------------------------*)
		IF st_ctrl_in.b_init THEN
			zyl_oelen_oben.st_ctrl.in.b_quittieren := FALSE;
			zyl_oelen_unten.st_ctrl.in.b_quittieren := FALSE;
			fb_state_entry.i16_next_step := 20;
		END_IF

(*=======================================================*)
	20: (* Abfrage Datum / Uhrzeit wegen Ölen nach Stillstand*)

		(*-----------------------Weiterschaltbedingungen----------------------------*)
		IF (gdt_system_time - dt_datum_uhrzeit_letzte_oelung) > t_delta_zeitraum THEN
			fb_ton_oelzeit.PT := st_oelerdaten.t_oelzeit_nach_stillstand;
			fb_state_entry.i16_next_step := 30;
		ELSE
			fb_state_entry.i16_next_step := BEREIT;
		END_IF

(*=======================================================*)
	30: (* Ölen nach Stillstand *)
		IF fb_state_entry.E THEN
			dt_datum_uhrzeit_letzte_oelung := gdt_system_time;	(* Merken, dass geölt wurde *)
			fb_ton_oelzeit.IN := TRUE;
			a_ventil_oben := TRUE;
			a_ventil_unten := TRUE;
		END_IF

		(*-----------------------Weiterschaltbedingungen----------------------------*)
		IF  fb_ton_oelzeit.Q THEN
			fb_ton_oelzeit.IN := FALSE;
			a_ventil_oben := FALSE;
			a_ventil_unten := FALSE;
			fb_state_entry.i16_next_step := BEREIT;
		END_IF

(*=======================================================
	40: (* Bandölen, abhängig von WKZ-Daten Zylinder ausfahren *)


	(*-----------------------Weiterschaltbedingungen----------------------------*)
		IF zyl_oelen_unten.fb.e_sensor1_ausgefahren AND
			 zyl_oelen_oben.fb.e_sensor1_ausgefahren THEN
			b_zyl_unten:= FALSE;
			b_zyl_oben:= FALSE;
			fb_state_entry.i16_next_step := 50;
		END_IF

(*=======================================================*)
	50: (* Bandölen, abhängig von WKZ-Daten Zylinder ausfahren *)


	(*-----------------------Weiterschaltbedingungen----------------------------*)
		IF zyl_oelen_unten.fb.e_sensor1_eingefahren AND
			 zyl_oelen_oben.fb.e_sensor1_eingefahren THEN
			fb_state_entry.i16_next_step := BEREIT;
		END_IF
=======================================================*)
	BEREIT:
		IF fb_state_entry.E THEN
			st_ctrl_out.b_bereit := TRUE;
		END_IF

		IF st_config.b_station_aktiv THEN
			(* Ölen *)
		(*	IF (gi16_betriebsart = AUTO OR gi16_betriebsart = TIPPEN) THEN
				IF	gst_datensatz.st_wkz.st_oeler.i16_intervall_bandoelen =0 THEN  (*bei Intervall 0 Dauerölen*)
					a_ventil_oben :=  fb_winkeltrigger.Q OR visu.b_handoelen OR b_ibn_handoelen;
					a_ventil_unten :=  fb_winkeltrigger.Q OR visu.b_handoelen OR b_ibn_handoelen;
				ELSE
					a_ventil_oben :=  visu.b_handoelen OR b_ibn_handoelen;
					a_ventil_unten :=  visu.b_handoelen OR b_ibn_handoelen;
				END_IF
			END_IF *)
			(* Überwachung Füllstand Betriebsmeldung*)
			IF NOT e_fuellstand AND e_steuerung_ein THEN
				bm_fuellstand_oeler := TRUE;
			ELSE
				bm_fuellstand_oeler := FALSE;
			END_IF
			(* Überwachung Füllstand Störmeldung *)
			IF fb_ton_uez_fuellstand.Q OR sm_fuellstand_oeler THEN
				sm_fuellstand_oeler := TRUE;
				st_ctrl_out.b_einzelfertigung:=TRUE;

				IF 	gi16_maschinenstatusinfo = STATUS_BETRIEBSBEREIT THEN
					fb_state_entry.i16_next_step := FEHLER;
				END_IF

			END_IF
			(* Überwachung Druck im Ölbehälter *)
			IF fb_ton_uez.Q OR sm_druckueberwachung THEN
				sm_druckueberwachung := TRUE;
				st_ctrl_out.b_einzelfertigung:=TRUE;

				IF 	gi16_maschinenstatusinfo = STATUS_BETRIEBSBEREIT THEN
					fb_state_entry.i16_next_step := FEHLER;
				END_IF
			END_IF

			(*-----------------------Weiterschaltbedingungen----------------------------*)
			IF	 i16_hubzaehler >= gst_datensatz.st_wkz.st_oeler.i16_intervall_bandoelen AND
				gst_datensatz.st_wkz.st_oeler.i16_intervall_bandoelen <>0 THEN (*bei Intervall 0 Dauerölen*)
				fb_state_entry.i16_next_step := 110;
			END_IF

		END_IF

(*=======================================================*)
	110: (* Bandölen, abhängig von WKZ-Daten Zylinder ausfahren *)
		IF fb_state_entry.E THEN
			dt_datum_uhrzeit_letzte_oelung := gdt_system_time;	(* Merken wann das letze mal geölt wurde *)
			i16_hubzaehler := 0;
			fb_ton_oelen.IN := TRUE;
			fb_ton_oelen.PT := DINT_TO_TIME(gst_datensatz.st_wkz.st_oeler.t_ventiloeffnungszeit);
			a_ventil_oben:= TRUE;
			a_ventil_unten:= TRUE;
		END_IF

		(*-----------------------Weiterschaltbedingungen----------------------------*)
		IF fb_ton_oelen.Q THEN
			fb_ton_oelen.IN := FALSE;
			a_ventil_oben := FALSE;
			a_ventil_unten := FALSE;
			fb_state_entry.i16_next_step := BEREIT;
		END_IF
(*=======================================================
	120: (* Bandölen, abhängig von WKZ-Daten Zylinder ausfahren *)


	(*-----------------------Weiterschaltbedingungen----------------------------*)
		IF zyl_oelen_unten.fb.e_sensor1_ausgefahren AND
			 zyl_oelen_oben.fb.e_sensor1_ausgefahren THEN
			b_zyl_unten:= FALSE;
			b_zyl_oben:= FALSE;
			fb_state_entry.i16_next_step := 130;
		END_IF

(*=======================================================*)
	130: (* Bandölen, abhängig von WKZ-Daten Zylinder ausfahren *)


	(*-----------------------Weiterschaltbedingungen----------------------------*)
		IF zyl_oelen_unten.fb.e_sensor1_eingefahren AND
			 zyl_oelen_oben.fb.e_sensor1_eingefahren THEN
			fb_state_entry.i16_next_step := BEREIT;
		END_IF
=======================================================*)
	FEHLER:
		IF fb_state_entry.E THEN
			st_ctrl_out.b_fehler := TRUE;
			a_ventil_oben := FALSE;
			a_ventil_unten := FALSE;
			fb_ton_quitt.IN := FALSE;
			zyl_oelen_oben.st_ctrl.in.b_quittieren := FALSE;
			zyl_oelen_unten.st_ctrl.in.b_quittieren := FALSE;
		END_IF

		(*-----------------------Weiterschaltbedingungen----------------------------*)
		IF st_ctrl_in.b_quitt AND NOT fb_state_entry.E THEN
			st_ctrl_out.b_fehler := FALSE;
			fb_ton_quitt.IN := TRUE;
			zyl_oelen_oben.st_ctrl.in.b_quittieren := TRUE;
			zyl_oelen_unten.st_ctrl.in.b_quittieren := TRUE;
		END_IF

		IF fb_ton_quitt.Q THEN
			fb_ton_quitt.IN := FALSE;
			fb_state_entry.i16_next_step := INIT;
		END_IF

(*=======================================================*)
	STOP:
		IF fb_state_entry.E THEN
			a_ventil_oben := FALSE;
			a_ventil_unten := FALSE;
			fb_ton_quitt.IN := FALSE;
			zyl_oelen_oben.st_ctrl.in.b_quittieren := FALSE;
			zyl_oelen_unten.st_ctrl.in.b_quittieren := FALSE;
		END_IF

		(*-----------------------Weiterschaltbedingungen----------------------------*)
		IF st_ctrl_in.b_quitt AND NOT fb_state_entry.E THEN
			fb_ton_quitt.IN := TRUE;
			zyl_oelen_oben.st_ctrl.in.b_quittieren := TRUE;
			zyl_oelen_unten.st_ctrl.in.b_quittieren := TRUE;
		END_IF

		IF fb_ton_quitt.Q THEN
			fb_ton_quitt.IN := FALSE;
			fb_state_entry.i16_next_step := INIT;
		END_IF
END_CASE

fb_state_entry(
	i16_next_step:= , 
	i16_pos:= 2,
	s_debugtext:= ,
	E=> ,
	X=> , 
	i16_step=> ,
	i16_last_step=> );

IF st_config.b_config_fertig THEN
	(* Fehlermeldungen und Betriebsmeldungen ab dem Startindex in die globalen Meldungsarrays schreiben *)
	garr_stoermeldungen[st_config.i16_meld_startindex + 0] := sm_fuellstand_oeler;
	garr_stoermeldungen[st_config.i16_meld_startindex + 1] := sm_druckueberwachung;
	garr_stoermeldungen[st_config.i16_meld_startindex + 2] := FALSE;
	garr_stoermeldungen[st_config.i16_meld_startindex + 3] := FALSE;
	garr_stoermeldungen[st_config.i16_meld_startindex + 4] := FALSE;
	garr_stoermeldungen[st_config.i16_meld_startindex + 5] := FALSE;
	garr_stoermeldungen[st_config.i16_meld_startindex + 6] := FALSE;
	garr_stoermeldungen[st_config.i16_meld_startindex + 7] := FALSE;
	garr_stoermeldungen[st_config.i16_meld_startindex + 8] := FALSE;
	garr_stoermeldungen[st_config.i16_meld_startindex + 9] := FALSE;
	garr_stoermeldungen[st_config.i16_meld_startindex + 10] := FALSE;
	garr_stoermeldungen[st_config.i16_meld_startindex + 11] := FALSE;
	garr_stoermeldungen[st_config.i16_meld_startindex + 12] := FALSE;
	garr_stoermeldungen[st_config.i16_meld_startindex + 13] := FALSE;
	garr_stoermeldungen[st_config.i16_meld_startindex + 14] := FALSE;
	garr_stoermeldungen[st_config.i16_meld_startindex + 15] := FALSE;
	garr_stoermeldungen[st_config.i16_meld_startindex + 16] := FALSE;
	garr_stoermeldungen[st_config.i16_meld_startindex + 17] := FALSE;
	garr_stoermeldungen[st_config.i16_meld_startindex + 18] := FALSE;
	garr_stoermeldungen[st_config.i16_meld_startindex + 19] := FALSE;
	
	garr_betriebsmeldungen[st_config.i16_meld_startindex + 0] := bm_fuellstand_oeler;
	garr_betriebsmeldungen[st_config.i16_meld_startindex + 1] := FALSE;
	garr_betriebsmeldungen[st_config.i16_meld_startindex + 2] := FALSE;
	garr_betriebsmeldungen[st_config.i16_meld_startindex + 3] := FALSE;
	garr_betriebsmeldungen[st_config.i16_meld_startindex + 4] := FALSE;
	garr_betriebsmeldungen[st_config.i16_meld_startindex + 5] := FALSE;
	garr_betriebsmeldungen[st_config.i16_meld_startindex + 6] := FALSE;
	garr_betriebsmeldungen[st_config.i16_meld_startindex + 7] := FALSE;
	garr_betriebsmeldungen[st_config.i16_meld_startindex + 8] := FALSE;
	garr_betriebsmeldungen[st_config.i16_meld_startindex + 9] := FALSE;
	garr_betriebsmeldungen[st_config.i16_meld_startindex + 10] := FALSE;
	garr_betriebsmeldungen[st_config.i16_meld_startindex + 11] := FALSE;
	garr_betriebsmeldungen[st_config.i16_meld_startindex + 12] := FALSE;
	garr_betriebsmeldungen[st_config.i16_meld_startindex + 13] := FALSE;
	garr_betriebsmeldungen[st_config.i16_meld_startindex + 14] := FALSE;
	garr_betriebsmeldungen[st_config.i16_meld_startindex + 15] := FALSE;
	garr_betriebsmeldungen[st_config.i16_meld_startindex + 16] := FALSE;
	garr_betriebsmeldungen[st_config.i16_meld_startindex + 17] := FALSE;
	garr_betriebsmeldungen[st_config.i16_meld_startindex + 18] := FALSE;
	garr_betriebsmeldungen[st_config.i16_meld_startindex + 19] := FALSE;
END_IF
END_PROGRAM

(* POU Gemeinsamkeiten17xx/TagReader/ST_Lesen_Schreiben_Tag, ST *)
PROGRAM ST_Lesen_Schreiben_Tag
VAR_INPUT
	st_config					: struct_config;
	st_ctrl_in					: struct_ctrl_in;
END_VAR
VAR_OUTPUT
	st_ctrl_out				: struct_ctrl_out;
END_VAR
VAR
	fb_r_trig_lesen			: R_TRIG;
	fb_r_trig_schreiben		: R_TRIG;
	fb_r_trig_WT_ruecksetzen	: R_TRIG;
	fb_r_trig_auto_lesen		: R_TRIG;
	fb_ton_lesen				: TON;
	fb_ton_auto_lesen				: TON;
	fb_ton_Timeout				: TON;

	fb_state_entry				: ST_StateEntry;
	fb_ton_quitt				: TON;
	fb_r_trig_quittieren			: R_TRIG;
	fb_ton_uez				: TON;

	sm_WT_Nummer_ungueltig				: BOOL := FALSE;
	sm_wt_hat_kein_tag					: BOOL := FALSE;
	bm_kein_WT_im_Aktionsfeld			: BOOL := FALSE;
	bm_Wert_nicht_erlaubt					: BOOL := FALSE;

	i									: INT;

	i16_betriebsart: BOOL;
END_VAR
fb_ton_quitt(IN:= , PT:= t#500ms, Q=> , ET=> );
fb_ton_uez(IN:= , PT:= , Q=>  , ET=> );

fb_ton_lesen(IN:= , PT:= t#500ms, Q=> , ET=> );
fb_r_trig_lesen(CLK:=visu.st_tagreader.b_start_lesen , Q=>);
fb_ton_auto_lesen(IN:=balluff_tag_reader.fb.e_tag_im_aktionsfeld   AND gi16_betriebsart = HAND , PT:= t#500ms, Q=> , ET=> );
fb_r_trig_auto_lesen(CLK:= fb_ton_auto_lesen.Q , Q=>);


fb_r_trig_schreiben(CLK:=visu.st_tagreader.b_start_schreiben , Q=>);
fb_r_trig_WT_ruecksetzen(CLK:=visu.st_tagreader.b_WT_ruecksetzen , Q=>);

visu.st_tagreader.b_tag_im_Aktionsfeld:=balluff_tag_reader.fb.e_tag_im_aktionsfeld;

fb_state_entry(
	i16_next_step:= ,
	i16_pos:= 1,
	s_debugtext:= ,
	E=> ,
	X=> ,
	i16_step=> ,
	i16_last_step=> );

(*wenn Tagreader nicht bereit ist stoppen*)
IF	Balluff_Tag_Reader.fb.fb_state_entry.i16_step<BEREIT OR
	Balluff_Tag_Reader.fb.fb_state_entry.i16_step>=STOP THEN
	fb_state_entry.i16_next_step := STOP;
END_IF

fb_ton_Timeout(IN:= fb_state_entry.i16_step>BEREIT AND fb_state_entry.i16_step<FEHLER, PT:= t#35s, Q=> , ET=> );
IF	fb_ton_Timeout.Q THEN
	fb_state_entry.i16_next_step := FEHLER;
END_IF

CASE fb_state_entry.i16_step OF
(*=======================================================*)
	INIT_OBJ:

		fb_state_entry.i16_next_step := INIT;

(*=======================================================*)
	INIT:
		IF 	fb_state_entry.E THEN
			balluff_tag_reader.st_ctrl.in.b_start_lesen := FALSE;
			balluff_tag_reader.st_ctrl.in.b_start_schreiben := FALSE;

			sm_WT_Nummer_ungueltig:=FALSE;
			sm_wt_hat_kein_tag:=FALSE;

			visu.st_tagreader.b_WT_ruecksetzen:=FALSE;
			visu.st_tagreader.b_start_schreiben:=FALSE;
			visu.st_tagreader.b_start_lesen:=FALSE;
		END_IF

		(*-----------------------Weiterschaltbedingungen----------------------------*)
		fb_state_entry.i16_next_step := BEREIT;

(*=======================================================*)
	BEREIT:	(* Warte auf Start von Kontroller *)

		(*-----------------------Weiterschaltbedingungen----------------------------*)
		IF	balluff_tag_reader.fb.e_tag_im_aktionsfeld   AND gi16_betriebsart = HAND THEN
			IF	fb_r_trig_lesen.Q  OR fb_r_trig_auto_lesen.Q THEN
				fb_state_entry.i16_next_step := 120;
			END_IF

			IF	fb_r_trig_schreiben.Q THEN
				fb_state_entry.i16_next_step := 150;
			END_IF

			IF	fb_r_trig_WT_ruecksetzen.Q THEN
				fb_state_entry.i16_next_step := 200;
			END_IF
		ELSE
			IF	fb_r_trig_WT_ruecksetzen.Q OR
				fb_r_trig_schreiben.Q OR
				fb_r_trig_lesen.Q THEN
				fb_state_entry.i16_next_step := 110;
			END_IF
		END_IF

(*=======================================================*)
	110:
		IF 	fb_state_entry.E THEN
			fb_ton_uez.PT:=t#2000ms ;
			fb_ton_uez.IN:=TRUE ;
			bm_kein_WT_im_Aktionsfeld:=TRUE;
		END_IF

		(*-----------------------Weiterschaltbedingungen----------------------------*)
		IF	fb_ton_uez.Q THEN
			fb_state_entry.i16_next_step := INIT;
			fb_ton_uez.IN:=FALSE ;
			bm_kein_WT_im_Aktionsfeld:=FALSE;
		END_IF

(*=======================================================*)
	120:
		IF 	fb_state_entry.E THEN
			gst_tag_data.Articelnumber:='LESEN';
			gst_tag_data.LastUsedTool:=0;
			IF gst_datensatz.st_md.i16_tag_data_structur_version = 0 THEN
				gst_tag_data.StateParts[0]:=100;
				gst_tag_data.StateParts[1]:=100;
			ELSIF gst_datensatz.st_md.i16_tag_data_structur_version = 1 THEN
				FOR i:= 0 TO 7 BY 1 DO
					gst_tag_data.StateParts[i] := 100;
				END_FOR
			END_IF
			gst_tag_data.WpcNumber:=0;
			fb_ton_lesen.IN:=TRUE;
		END_IF

	(*-----------------------Weiterschaltbedingungen----------------------------*)
	IF	fb_ton_lesen.Q THEN
		fb_ton_lesen.IN:=FALSE;
		fb_state_entry.i16_next_step := 130;
	END_IF

(*=======================================================*)
	130: (* WT-Tag mit RFID-Lesegerät auslesen *)
		IF 	fb_state_entry.E THEN
			balluff_tag_reader.st_ctrl.in.b_start_lesen := TRUE;
			balluff_tag_reader.fb.i16_addresse := 0;
			balluff_tag_reader.fb.i16_anzahl_byte := SIZEOF(gst_tag_data);
		END_IF

		(*-----------------------Weiterschaltbedingungen----------------------------*)
		IF 	balluff_tag_reader.st_ctrl.out.b_fertig AND NOT fb_state_entry.E THEN
			IF gst_datensatz.st_md.i16_tag_data_structur_version = 0 THEN
				gst_tag_data.WpcNumber := balluff_tag_reader.fb.s_lese_daten[0];
				gst_tag_data.StateParts[0] := balluff_tag_reader.fb.s_lese_daten[1];
				gst_tag_data.StateParts[1] := balluff_tag_reader.fb.s_lese_daten[2];

				MEMCPY( ADR(gst_tag_data.Articelnumber), ADR(balluff_tag_reader.fb.s_lese_daten[3]), 50);
				gst_tag_data.LastUsedTool := balluff_tag_reader.fb.s_lese_daten[54];
				MEMCPY( ADR(gst_tag_data.UmlNo_VPE), ADR(balluff_tag_reader.fb.s_lese_daten[55]), 4);

				(*gst_datensatz.st_md.s_aktuelle_artikelnummer := gst_tag_data.Articelnumber;*)
			ELSIF gst_datensatz.st_md.i16_tag_data_structur_version = 1 THEN
				gst_tag_data.WpcNumber := balluff_tag_reader.fb.s_lese_daten[0];
				FOR i:= 0 TO 7 BY 1 DO
					gst_tag_data.StateParts[i] := balluff_tag_reader.fb.s_lese_daten[i + 1];
				END_FOR
				gst_tag_data.AmountPartsOnWpc := balluff_tag_reader.fb.s_lese_daten[10];
				gst_tag_data.LastUsedTool := balluff_tag_reader.fb.s_lese_daten[15];
				MEMCPY( ADR(gst_tag_data.Articelnumber), ADR(balluff_tag_reader.fb.s_lese_daten[20]), 50);
				MEMCPY( ADR(gst_tag_data.UmlNo_VPE), ADR(balluff_tag_reader.fb.s_lese_daten[71]), 4);
			END_IF

			IF 	gst_tag_data.WpcNumber >= 0 AND gst_tag_data.WpcNumber <=50 THEN
				balluff_tag_reader.st_ctrl.in.b_start_lesen := FALSE;
				fb_state_entry.i16_next_step := INIT;
			ELSE
				(* Fehler: Tagnummer ist nicht im gültigem Bereich *)
				balluff_tag_reader.st_ctrl.in.b_start_lesen := FALSE;
				sm_WT_Nummer_ungueltig := TRUE;
				fb_state_entry.i16_next_step := FEHLER;
			END_IF
		END_IF

(*=======================================================*)
	150:	(*Artikelnummer schreiben*)
		IF 	fb_state_entry.E THEN
			IF gst_datensatz.st_md.i16_tag_data_structur_version = 0 THEN
				balluff_tag_reader.st_ctrl.in.b_start_schreiben := TRUE;
	
				balluff_tag_reader.fb.i16_addresse := 3;
				balluff_tag_reader.fb.i16_anzahl_byte := SIZEOF(gst_tag_data.Articelnumber);
				MEMCPY(ADR(balluff_tag_reader.fb.s_schreib_daten),ADR(gst_tag_data.Articelnumber),  50);
			ELSIF gst_datensatz.st_md.i16_tag_data_structur_version = 1 THEN
				balluff_tag_reader.st_ctrl.in.b_start_schreiben := TRUE;
	
				balluff_tag_reader.fb.i16_addresse := 20;
				balluff_tag_reader.fb.i16_anzahl_byte := SIZEOF(gst_tag_data.Articelnumber);
				MEMCPY(ADR(balluff_tag_reader.fb.s_schreib_daten),ADR(gst_tag_data.Articelnumber),  50);
			END_IF
		END_IF

		(*-----------------------Weiterschaltbedingungen----------------------------*)
		IF 	balluff_tag_reader.st_ctrl.out.b_fertig AND NOT fb_state_entry.E THEN
			(* Ok: Daten sind auf dem Tag *)
			balluff_tag_reader.st_ctrl.in.b_start_schreiben := FALSE;
			fb_state_entry.i16_next_step := 155;
		END_IF

(*=======================================================*)
	155:	(*UML_Stueckzaehler schreiben*)
		IF 	fb_state_entry.E THEN
			IF gst_datensatz.st_md.i16_tag_data_structur_version = 0 THEN
				balluff_tag_reader.st_ctrl.in.b_start_schreiben := TRUE;

				balluff_tag_reader.fb.i16_addresse := 55;
				balluff_tag_reader.fb.i16_anzahl_byte := SIZEOF(gst_tag_data.UmlNo_VPE);
				MEMCPY( ADR(balluff_tag_reader.fb.s_schreib_daten), ADR(gst_tag_data.UmlNo_VPE), 4);

			ELSIF gst_datensatz.st_md.i16_tag_data_structur_version = 1 THEN
				balluff_tag_reader.st_ctrl.in.b_start_schreiben := TRUE;

				balluff_tag_reader.fb.i16_addresse := 71;
				balluff_tag_reader.fb.i16_anzahl_byte := SIZEOF(gst_tag_data.UmlNo_VPE);
				MEMCPY(ADR(balluff_tag_reader.fb.s_schreib_daten),ADR(gst_tag_data.UmlNo_VPE),  4);
			END_IF
		END_IF

		(*-----------------------Weiterschaltbedingungen----------------------------*)
		IF 	balluff_tag_reader.st_ctrl.out.b_fertig AND NOT fb_state_entry.E THEN
			(* Ok: Daten sind auf dem Tag *)
			balluff_tag_reader.st_ctrl.in.b_start_schreiben := FALSE;
			fb_state_entry.i16_next_step := 160;
		END_IF

(*=======================================================*)
	160:	(*States schreiben*)
		IF 	fb_state_entry.E THEN
			IF gst_datensatz.st_md.i16_tag_data_structur_version = 0 THEN
				balluff_tag_reader.st_ctrl.in.b_start_schreiben := TRUE;
	
				balluff_tag_reader.fb.i16_addresse := 1;
				balluff_tag_reader.fb.i16_anzahl_byte := 2;
				balluff_tag_reader.fb.s_schreib_daten[0] := DINT_TO_BYTE(gst_tag_data.StateParts[0]);
				balluff_tag_reader.fb.s_schreib_daten[1] := DINT_TO_BYTE(gst_tag_data.StateParts[1]);
			ELSIF gst_datensatz.st_md.i16_tag_data_structur_version = 1 THEN
				balluff_tag_reader.st_ctrl.in.b_start_schreiben := TRUE;
	
				balluff_tag_reader.fb.i16_addresse := 1;
				balluff_tag_reader.fb.i16_anzahl_byte := 8;
				FOR i:= 0 TO 7 BY 1 DO
					balluff_tag_reader.fb.s_schreib_daten[i] := DINT_TO_BYTE(gst_tag_data.StateParts[i]);
				END_FOR
			END_IF
		END_IF

		(*-----------------------Weiterschaltbedingungen----------------------------*)
		IF balluff_tag_reader.st_ctrl.out.b_fertig AND NOT fb_state_entry.E THEN
			(* Ok: Daten sind auf dem Tag *)
			balluff_tag_reader.st_ctrl.in.b_start_schreiben := FALSE;
			fb_state_entry.i16_next_step := 170;
		END_IF

